# B&R Automation Studio project A2019059_Linka_Power_CP (part 12)

#### Axis_Krokac.st
```iecst
(* TODO: Add your comment here *)
FUNCTION_BLOCK Axis_Krokac

	//***********************************************************Power krokáča*********************************************************************//
	Internal.MC_Power_0.Axis:= AxisName;
	Internal.MC_Power_0.Enable:= CMD.POWER;
	ErrorDetail.Power_Error:= Internal.MC_Power_0.Error;
	ErrorDetail.Power_ErrorID:= Internal.MC_Power_0.ErrorID;
	Internal.MC_Power_0();

	//***********************************************************Zobrazenie stavu krokáča*********************************************************//
	Internal.MC_ReadAxisInfo_0.Axis:= AxisName;
	Internal.MC_ReadAxisInfo_0.Enable:= TRUE;
	STATUS.ReadyToPower_ON := Internal.MC_ReadAxisInfo_0.ReadyForPowerOn;
	STATUS.Communication_READY:= Internal.MC_ReadAxisInfo_0.CommunicationReady;
	STATUS.Power_ON:= Internal.MC_ReadAxisInfo_0.PowerOn;
	STATUS.Homing_OK:= Internal.MC_ReadAxisInfo_0.IsHomed;
	STATUS.EnableSwitch_ACTIVE:= Internal.MC_ReadAxisInfo_0.AdditionalInfo.DigitalInputStatus.DriveEnable;
	STATUS.HomingSwitch_ACTIVE:= Internal.MC_ReadAxisInfo_0.AdditionalInfo.DigitalInputStatus.HomingSwitch;
	STATUS.NegativeLimitSwitch_ACTIVE:=	Internal.MC_ReadAxisInfo_0.AdditionalInfo.DigitalInputStatus.NegativeLimitSwitch;
	STATUS.PositiveLimitSwitch_ACTIVE:=	Internal.MC_ReadAxisInfo_0.AdditionalInfo.DigitalInputStatus.PositiveLimitSwitch;
	Internal.MC_ReadAxisInfo_0();

	//********************************************************Porucha krokáča************************************************************************//
	//Zobrazenie poruchy krokáča//
	Internal.MC_ReadAxisError_0.Axis:= AxisName;
	Internal.MC_ReadAxisError_0.Enable:= CMD.ENABLE;
	STATUS.ERROR_ID:= Internal.MC_ReadAxisError_0.AxisErrorID;
	Internal.MC_ReadAxisError_0();

	Internal.MC_ReadStatus_0.Axis:= AxisName;
	Internal.MC_ReadStatus_0.Enable:= CMD.ENABLE;
	Internal.MC_ReadStatus_0();

	IF Internal.MC_Power_0.Error THEN
		STATUS.ERROR:= TRUE;
	ELSIF Internal.MC_Home_0.Error THEN
		STATUS.ERROR:= TRUE;
	ELSIF Internal.MC_BR_JogLimitPosition_0.Error THEN
		STATUS.ERROR:= TRUE;
	ELSIF Internal.MC_BR_JogVelocity_0.Error THEN
		STATUS.ERROR:= TRUE;
	ELSIF Internal.MC_MoveAbsolute_0.Error THEN
		STATUS.ERROR:= TRUE;
	ELSIF Internal.MC_MoveAdditive_0.Error THEN
		STATUS.ERROR:= TRUE;
	ELSIF Internal.MC_MoveVelocity_0.Error THEN
		STATUS.ERROR:= TRUE;
	ELSIF Internal.MC_Stop_0.Error THEN
		STATUS.ERROR:= TRUE;
	ELSIF Internal.MC_BR_BrakeOperation_0.Error THEN
		STATUS.ERROR:= TRUE;
	ELSIF Internal.MC_BR_InitHome_StpAx_0.Error THEN
		STATUS.ERROR:= TRUE;
	ELSIF STATUS.ERROR_ID <> 0 THEN
		STATUS.ERROR:= TRUE;
	ELSE
		STATUS.ERROR:= FALSE;
	END_IF

	//Reset poruchy krokáča//
	Internal.MC_Reset_0.Axis:= AxisName;
	Internal.MC_Reset_0.Execute:= CMD.ErrorRESET;
	Internal.MC_Reset_0();

	IF CMD.ErrorRESET THEN
		CMD.ENABLE:= FALSE;
	ELSE
		CMD.ENABLE:= TRUE;
	END_IF

	//*********************************************Homing krokáča***************************************************************************//
	//Parametre homingu//
	Internal.MC_BR_InitHome_StpAx_0.Axis:= AxisName;
	Internal.MC_Home_0.Axis:= AxisName;
	IF HomePAR.HomingMode = 0 THEN //Homing na mieste
		Internal.MC_BR_InitHome_StpAx_0.HomingParameters.HomingMode:= mcHOMING_DIRECT;
	ELSIF HomePAR.HomingMode = 1 THEN //Homing na refernčný snímač
		Internal.MC_BR_InitHome_StpAx_0.HomingParameters.HomingMode:= mcHOMING_SWITCH_GATE;
		Internal.MC_BR_InitHome_StpAx_0.HomingParameters.StartDirection:= mcDIR_NEGATIVE;  //Smer hladania refernčného snímača
		Internal.MC_BR_InitHome_StpAx_0.HomingParameters.SwitchEdge:= mcDIR_NEGATIVE; //Typ hrany referenčného snímača
		Internal.MC_BR_InitHome_StpAx_0.HomingParameters.HomingDirection:= mcDIR_POSITIVE; //Smer odchodu z referenčného snímača
	ELSIF HomePAR.HomingMode = 2 THEN //Homing na limitný snímač
		Internal.MC_BR_InitHome_StpAx_0.HomingParameters.HomingMode:= mcHOMING_LIMIT_SWITCH;
		Internal.MC_BR_InitHome_StpAx_0.HomingParameters.SwitchEdge:= mcDIR_NEGATIVE; //Typ hrany referenčného snímača
		Internal.MC_BR_InitHome_StpAx_0.HomingParameters.HomingDirection:= mcDIR_POSITIVE; //Smer odchodu z referenčného snímača
	ELSE
		Internal.MC_BR_InitHome_StpAx_0.HomingParameters.HomingMode:= mcHOMING_DIRECT;
	END_IF
	Internal.MC_BR_InitHome_StpAx_0.HomingParameters.Acceleration:= HomePAR.Acceleration;
	Internal.MC_BR_InitHome_StpAx_0.HomingParameters.HomingVelocity:= HomePAR.HomingVelocity;
	Internal.MC_BR_InitHome_StpAx_0.HomingParameters.Position:= HomePAR.Position;
	Internal.MC_BR_InitHome_StpAx_0.HomingParameters.StartVelocity:= HomePAR.StartVelocity;
	Internal.MC_BR_InitHome_StpAx_0.HomingParameters.ReferencePulse:= mcSWITCH_OFF;
	Internal.MC_BR_InitHome_StpAx_0.HomingParameters.KeepDirection:= mcSWITCH_OFF;
	Internal.MC_Home_0.HomingMode:= mcHOMING_INIT;
	Internal.MC_Home_0.BufferMode:= mcABORTING;
	STATUS.Homing_BUSY:= Internal.MC_Home_0.Busy;
	ErrorDetail.Home_Error:= Internal.MC_Home_0.Error;
	ErrorDetail.Home_ErrorID:= Internal.MC_Home_0.ErrorID;
	Internal.MC_BR_InitHome_StpAx_0();
	Internal.MC_Home_0();

	CASE Internal.Home_STEP OF

		0: //Nulovanie//
			Internal.MC_BR_InitHome_StpAx_0.Execute:= FALSE;
			Internal.MC_Home_0.Execute:= FALSE;
			IF NOT CMD.HOME AND NOT Internal.MC_BR_InitHome_StpAx_0.Error AND NOT Internal.MC_Home_0.Error THEN
				Internal.Home_STEP:= 1;
			END_IF

		1: //Čakanie na spustenie homingu//
			IF CMD.HOME THEN
				Internal.Home_STEP:= 2;
			END_IF

		2: //Načítanie parametrov homingu//
			Internal.MC_BR_InitHome_StpAx_0.Execute:= TRUE;
			IF Internal.MC_BR_InitHome_StpAx_0.Error THEN
				Internal.Home_STEP:= 0;
			ELSIF Internal.MC_BR_InitHome_StpAx_0.Done THEN
				Internal.MC_BR_InitHome_StpAx_0.Execute:= FALSE;
				Internal.Home_STEP:= 3;
			END_IF

		3: //Spustenie homingu
			Internal.MC_Home_0.Execute:= TRUE;
			IF Internal.MC_Home_0.Error THEN
				Internal.Home_STEP:= 0;
			ELSIF Internal.MC_Home_0.Done THEN
				Internal.Home_STEP:= 0;
			ELSIF NOT CMD.HOME THEN
				Internal.Home_STEP:= 0;
			END_IF
	END_CASE

	//*********************************************Jogging krokáča**************************************************************************//

	IF (CMD.JoggVPRED OR CMD.JoggVZAD) AND NOT CMD.JoggLimit_ACTIVE AND CMD.ENABLE THEN
		Internal.MC_BR_JogLimitPosition_0.Enable:= FALSE;
		Internal.MC_BR_JogVelocity_0.Enable:= TRUE;
		STATUS.Jogging_BUSY:= Internal.MC_BR_JogVelocity_0.Jogging;
	ELSIF (CMD.JoggVPRED OR CMD.JoggVZAD) AND CMD.JoggLimit_ACTIVE AND CMD.ENABLE THEN
		Internal.MC_BR_JogVelocity_0.Enable:= FALSE;
		Internal.MC_BR_JogLimitPosition_0.Enable:= TRUE;
		STATUS.Jogging_BUSY:= Internal.MC_BR_JogLimitPosition_0.Jogging;
	ELSE
		Internal.MC_BR_JogVelocity_0.Enable:= FALSE;
		Internal.MC_BR_JogLimitPosition_0.Enable:= FALSE;
	END_IF

	//Normálny jogg//
	Internal.MC_BR_JogVelocity_0.Axis:= AxisName;
	Internal.MC_BR_JogVelocity_0.Acceleration:= PAR.JoggAcceleration;
	Internal.MC_BR_JogVelocity_0.Deceleration:= PAR.JoggDeceleration;
	Internal.MC_BR_JogVelocity_0.Velocity:= PAR.JoggVelocity;
	Internal.MC_BR_JogVelocity_0.Jerk:= 0.0;
	Internal.MC_BR_JogVelocity_0.JogPositive:= CMD.JoggVPRED;
	Internal.MC_BR_JogVelocity_0.JogNegative:= CMD.JoggVZAD;
	ErrorDetail.Jogg_Error:= Internal.MC_BR_JogVelocity_0.Error;
	ErrorDetail.Jogg_ErrorID:= Internal.MC_BR_JogVelocity_0.ErrorID;
	Internal.MC_BR_JogVelocity_0();

	//Limitný jogg//
	Internal.MC_BR_JogLimitPosition_0.Axis:= AxisName;
	IF STATUS.ActualPosition >= PAR.JoggPoziciaLimitVPRED THEN
		Internal.MC_BR_JogLimitPosition_0.LastPosition:= STATUS.ActualPosition;
	ELSE
		Internal.MC_BR_JogLimitPosition_0.LastPosition:= PAR.JoggPoziciaLimitVPRED;
	END_IF
	IF STATUS.ActualPosition <= PAR.JoggPoziciaLimitVZAD THEN
		Internal.MC_BR_JogLimitPosition_0.FirstPosition:= STATUS.ActualPosition;
	ELSE
		Internal.MC_BR_JogLimitPosition_0.FirstPosition:= PAR.JoggPoziciaLimitVZAD;
	END_IF
	Internal.MC_BR_JogLimitPosition_0.Acceleration:= PAR.JoggAcceleration;
	Internal.MC_BR_JogLimitPosition_0.Deceleration:= PAR.JoggDeceleration;
	Internal.MC_BR_JogLimitPosition_0.Jerk:= 0.0;
	Internal.MC_BR_JogLimitPosition_0.JogPositive:= CMD.JoggVPRED;
	Internal.MC_BR_JogLimitPosition_0.JogNegative:= CMD.JoggVZAD;
	Internal.MC_BR_JogLimitPosition_0.Velocity:= PAR.JoggVelocity;
	STATUS.JoggLimit_Dosiahnuty:= Internal.MC_BR_JogLimitPosition_0.LimitReached;
	ErrorDetail.JoggLimit_Error:= Internal.MC_BR_JogLimitPosition_0.Error;
	ErrorDetail.JoggLimit_ErrorID:= Internal.MC_BR_JogLimitPosition_0.ErrorID;
	Internal.MC_BR_JogLimitPosition_0();

	//********************************************Move Absolute***************************************************************************//
	Internal.MC_MoveAbsolute_0.Axis:= AxisName;
	Internal.MC_MoveAbsolute_0.Execute:= CMD.MoveAbsolute;
	Internal.MC_MoveAbsolute_0.Acceleration:= PAR.Acceleration;
	Internal.MC_MoveAbsolute_0.Deceleration:= PAR.Deceleration;
	Internal.MC_MoveAbsolute_0.BufferMode:= mcABORTING;
	IF PAR.MoveDirection = 0 THEN
		Internal.MC_MoveAbsolute_0.Direction:= mcDIR_POSITIVE;
	ELSIF PAR.MoveDirection = 1 THEN
		Internal.MC_MoveAbsolute_0.Direction:= mcDIR_NEGATIVE;
	ELSIF PAR.MoveDirection = 10 THEN
		Internal.MC_MoveAbsolute_0.Direction:= mcDIR_BOTH;
	ELSE
		Internal.MC_MoveAbsolute_0.Direction:= 0;
	END_IF
	Internal.MC_MoveAbsolute_0.Jerk:= 0.0;
	Internal.MC_MoveAbsolute_0.Position:= PAR.Position;
	Internal.MC_MoveAbsolute_0.Velocity:= PAR.Velocity;
	STATUS.MoveAbsolute_BUSY:= Internal.MC_MoveAbsolute_0.Busy;
	STATUS.MoveAbsolute_DONE:= Internal.MC_MoveAbsolute_0.Done;
	ErrorDetail.MoveAbsolute_Error:= Internal.MC_MoveAbsolute_0.Error;
	ErrorDetail.MoveAbsolute_ErrorID:= Internal.MC_MoveAbsolute_0.ErrorID;
	Internal.MC_MoveAbsolute_0();

	//********************************************Move Additive*****************************************************************************//
	Internal.MC_MoveAdditive_0.Axis:= AxisName;
	Internal.MC_MoveAdditive_0.Execute:= CMD.MoveAdditive;
	Internal.MC_MoveAdditive_0.Acceleration:= PAR.Acceleration;
	Internal.MC_MoveAdditive_0.Deceleration:= PAR.Deceleration;
	Internal.MC_MoveAdditive_0.Distance:= PAR.AdditivePosition;
	Internal.MC_MoveAdditive_0.Velocity:= PAR.Velocity;
	Internal.MC_MoveAdditive_0.BufferMode:= mcABORTING;
	Internal.MC_MoveAdditive_0.Jerk:= 0.0;
	STATUS.MoveAdditive_BUSY:= Internal.MC_MoveAdditive_0.Busy;
	STATUS.MoveAdditive_DONE:= Internal.MC_MoveAdditive_0.Done;
	ErrorDetail.MoveAdditive_Error:= Internal.MC_MoveAdditive_0.Error;
	ErrorDetail.MoveAdditive_ErrorID:= Internal.MC_MoveAdditive_0.ErrorID;
	Internal.MC_MoveAdditive_0();

	//*********************************************Move Velocity****************************************************************************//
	Internal.MC_MoveVelocity_0.Axis:= AxisName;
	Internal.MC_MoveVelocity_0.Execute:= CMD.MoveVelocity;
	Internal.MC_MoveVelocity_0.Acceleration:= PAR.Acceleration;
	Internal.MC_MoveVelocity_0.Deceleration:= PAR.Deceleration;
	Internal.MC_MoveVelocity_0.BufferMode:= mcABORTING;
	IF PAR.MoveDirection = 0 THEN
		Internal.MC_MoveVelocity_0.Direction:= mcDIR_POSITIVE;
	ELSIF PAR.MoveDirection = 1 THEN
		Internal.MC_MoveVelocity_0.Direction:= mcDIR_NEGATIVE;
	ELSIF PAR.MoveDirection = 10 THEN
		Internal.MC_MoveVelocity_0.Direction:= mcDIR_BOTH;
	ELSE
		Internal.MC_MoveVelocity_0.Direction:= 0;
	END_IF
	Internal.MC_MoveVelocity_0.Velocity:= PAR.Velocity;
	Internal.MC_MoveVelocity_0.Jerk:= 0.0;
	STATUS.MoveVelocity_BUSY:= Internal.MC_MoveVelocity_0.Busy;
	STATUS.Rychlost_Dosiahnuta:= Internal.MC_MoveVelocity_0.InVelocity;
	ErrorDetail.MoveVelocity_Error:= Internal.MC_MoveVelocity_0.Error;
	ErrorDetail.MoveVelocity_ErrorID:= Internal.MC_MoveVelocity_0.ErrorID;
	Internal.MC_MoveVelocity_0();

	//********************************************Stop krokáča******************************************************************************//
	Internal.MC_Stop_0.Axis:= AxisName;
	Internal.MC_Stop_0.Execute:= CMD.STOP;
	Internal.MC_Stop_0.Deceleration:= PAR.StopDeceleration;
	Internal.MC_Stop_0.Jerk:= 0.0;
	STATUS.STOP_ACTIVE:= Internal.MC_Stop_0.Done;
	ErrorDetail.Stop_Error:= Internal.MC_Stop_0.Error;
	ErrorDetail.Stop_ErrorID:= Internal.MC_Stop_0.ErrorID;
	Internal.MC_Stop_0();

	//**********************************************Ovládanie brzdy************************************************************************//
	Internal.MC_BR_BrakeOperation_0.Axis:= AxisName;
	IF CMD.UvolniBRZDU THEN
		Internal.MC_BR_BrakeOperation_0.Command:= mcBRAKE_OPEN;
		Internal.MC_BR_BrakeOperation_0.Execute:= TRUE;
		STATUS.UvolnenieBrzdy_DONE:= Internal.MC_BR_BrakeOperation_0.Done;
	ELSIF CMD.ZabrzdiBRZDU THEN
		Internal.MC_BR_BrakeOperation_0.Command:= mcBRAKE_CLOSE;
		Internal.MC_BR_BrakeOperation_0.Execute:= TRUE;
		STATUS.ZabrzdenieBrzdy_DONE:= Internal.MC_BR_BrakeOperation_0.Done;
	ELSE
		Internal.MC_BR_BrakeOperation_0.Execute:= FALSE;
		STATUS.UvolnenieBrzdy_DONE:= FALSE;
		STATUS.ZabrzdenieBrzdy_DONE:= FALSE;
	END_IF
	ErrorDetail.BreakOperation_Error:= Internal.MC_BR_BrakeOperation_0.Error;
	ErrorDetail.BreakOperation_ErrorID:= Internal.MC_BR_BrakeOperation_0.ErrorID;
	Internal.MC_BR_BrakeOperation_0();

	//**********************************************Aktuálna pozícia*************************************************************************//
	Internal.MC_ReadActualPosition_0.Axis:= AxisName;
	Internal.MC_ReadActualPosition_0.Enable:= CMD.ENABLE;
	STATUS.ActualPosition:=	Internal.MC_ReadActualPosition_0.Position;
	Internal.MC_ReadActualPosition_0();

	//**********************************************Aktuálna rýchlosť*************************************************************************//
	Internal.MC_ReadActualVelocity_0.Axis:= AxisName;
	Internal.MC_ReadActualVelocity_0.Enable:= CMD.ENABLE;
	STATUS.ActualVelocity:= Internal.MC_ReadActualVelocity_0.Velocity;
	Internal.MC_ReadActualVelocity_0();

	//*********************************************Zmena rýchlosti a rampy********************************************************************//
	Internal.MC_SetOverride_0.Axis:= AxisName;
	Internal.MC_SetOverride_0.Enable:= CMD.UpdatePAR;
	IF PAR.ZmenaRampy < 0.1 THEN
		Internal.MC_SetOverride_0.AccFactor:= 0.1;
	ELSIF PAR.ZmenaRampy > 2.0 THEN
		Internal.MC_SetOverride_0.AccFactor:= 2.0;
	ELSE
		Internal.MC_SetOverride_0.AccFactor:= PAR.ZmenaRampy;
	END_IF
	IF PAR.ZmenaRychlosti < 0.1 THEN
		Internal.MC_SetOverride_0.VelFactor:= 0.1;
	ELSIF PAR.ZmenaRychlosti > 2.0 THEN
		Internal.MC_SetOverride_0.VelFactor:= 2.0;
	ELSE
		Internal.MC_SetOverride_0.VelFactor:= PAR.ZmenaRychlosti;
	END_IF
	STATUS.UpdatePAR_DONE:= Internal.MC_SetOverride_0.Enabled;
	Internal.MC_SetOverride_0();

END_FUNCTION_BLOCK
```

#### ServoLim.st
```iecst
(* TODO: Add your comment here *)
FUNCTION_BLOCK ServoLim

	//*******************************Aktivácia limitných snímačov*****************************************//
	//Reset poruchy//
	IF NOT ENABLE THEN
		Internal.STEP:= 0;
		Error:= FALSE;
	END_IF

	//Zápis do parametrov//

	CASE Internal.STEP OF

		0: //Čakanie na spustenie sekvencie//
			Internal.MC_BR_ProcessParID_AcpAx_0.Execute:= FALSE;
			Internal.MC_BR_CyclicProcessParID_AcpAx_0.Enable:= FALSE;
			BUSY:= FALSE;
			IF ENABLE AND NOT Error THEN
				Internal.STEP:= 1;
			END_IF

		1://Zápis parametru - povolenie limitných snímačov//
			Internal.MC_BR_ProcessParID_AcpAx_0.Axis:= AxisName;
			Internal.MC_BR_ProcessParID_AcpAx_0.DataAddress:= ADR(Internal.McAcpAxProcessParIDType_0);
			Internal.MC_BR_ProcessParID_AcpAx_0.NumberOfParIDs:= 0;
			Internal.MC_BR_ProcessParID_AcpAx_0.Mode:= mcACPAX_PARID_SET;
			Internal.McAcpAxProcessParIDType_0.DataType:= mcACPAX_PARTYPE_USINT;
			Internal.McAcpAxProcessParIDType_0.ParID:= 184;
			Internal.McAcpAxProcessParIDType_0.VariableAddress:= ADR(Internal.AktivaciaLimSnimacov_Data);
			Internal.AktivaciaLimSnimacov_Data:= 7;
			Internal.MC_BR_ProcessParID_AcpAx_0.Execute:= TRUE;

			IF Internal.MC_BR_ProcessParID_AcpAx_0.Done THEN
				Internal.MC_BR_ProcessParID_AcpAx_0.Execute:= FALSE;
				Internal.AktivaciaLimSnimacov_Data:= 0;
				Internal.STEP:= 3;
			ELSIF Internal.MC_BR_ProcessParID_AcpAx_0.Error THEN
				Error:= TRUE;
				Internal.STEP:= 0;
			END_IF

		3://Korekčný čas//
			IF NOT Internal.MC_BR_ProcessParID_AcpAx_0.Done THEN
				Internal.KorekcnyCas.IN:= TRUE;
			END_IF

			IF Internal.KorekcnyCas.Q THEN
				Internal.KorekcnyCas.IN:= FALSE;
				Internal.STEP:= 5;
			END_IF

		5://Čítanie parametru - overenie povolenia limitných snímačov//
			Internal.MC_BR_ProcessParID_AcpAx_0.Axis:= AxisName;
			Internal.MC_BR_ProcessParID_AcpAx_0.DataAddress:= ADR(Internal.McAcpAxProcessParIDType_0);
			Internal.MC_BR_ProcessParID_AcpAx_0.NumberOfParIDs:= 0;
			Internal.MC_BR_ProcessParID_AcpAx_0.Mode:= mcACPAX_PARID_GET;
			Internal.McAcpAxProcessParIDType_0.DataType:= mcACPAX_PARTYPE_USINT;
			Internal.McAcpAxProcessParIDType_0.ParID:= 184;
			Internal.McAcpAxProcessParIDType_0.VariableAddress:= ADR(Internal.AktivaciaLimSnimacov_Data);
			Internal.MC_BR_ProcessParID_AcpAx_0.Execute:= TRUE;

			IF Internal.MC_BR_ProcessParID_AcpAx_0.Done THEN
				IF Internal.AktivaciaLimSnimacov_Data = 7 THEN
					Internal.MC_BR_ProcessParID_AcpAx_0.Execute:= FALSE;
					Internal.STEP:= 10;
				ELSE
					Error:= TRUE;
					Internal.STEP:= 0;
				END_IF
			ELSIF Internal.MC_BR_ProcessParID_AcpAx_0.Error THEN
				Error:= TRUE;
				Internal.STEP:= 0;
			END_IF

		8://Korekčný čas//
			IF NOT Internal.MC_BR_ProcessParID_AcpAx_0.Done THEN
				Internal.KorekcnyCas.IN:= TRUE;
			END_IF

			IF Internal.KorekcnyCas.Q THEN
				Internal.KorekcnyCas.IN:= FALSE;
				Internal.STEP:= 10;
			END_IF

		10://
			Internal.MC_BR_CyclicProcessParID_AcpAx_0.Axis:= AxisName;
			Internal.MC_BR_CyclicProcessParID_AcpAx_0.DataAddress:= ADR(Internal.McAcpAxCycParIDType_0);
			Internal.MC_BR_CyclicProcessParID_AcpAx_0.NumberOfParIDs:= 0;
			Internal.MC_BR_CyclicProcessParID_AcpAx_0.Mode:= mcACPAX_CYCLIC_PARID_WRITE;
			Internal.McAcpAxCycParIDType_0.DataType:= mcACPAX_PARTYPE_USINT;
			Internal.McAcpAxCycParIDType_0.ParID:= 185;
			Internal.McAcpAxCycParIDType_0.VariableAddress:= ADR(Internal.LimSnimace_Data);
			Internal.McAcpAxCycParIDType_0.RefreshMode:= mcACPAX_CYCLIC_EVERY_RECORD;
			Internal.MC_BR_CyclicProcessParID_AcpAx_0.Enable:= TRUE;
			Internal.LimSnimace_Data.0:= HomingSwitch;
			Internal.LimSnimace_Data.1:= PositiveLimitSwitch;
			Internal.LimSnimace_Data.2:= NegativeLimitSwitch;

			BUSY:= Internal.MC_BR_CyclicProcessParID_AcpAx_0.Busy;

			IF Internal.MC_BR_CyclicProcessParID_AcpAx_0.Error THEN
				Error:= TRUE;
				Internal.STEP:= 0;
			END_IF

	END_CASE

	Internal.MC_BR_ProcessParID_AcpAx_0();
	Internal.MC_BR_CyclicProcessParID_AcpAx_0();

	Internal.KorekcnyCas.PT:= T#200ms;
	Internal.KorekcnyCas();

END_FUNCTION_BLOCK
```

### Library Logical/Libraries/IecCheck (IEC)
Depends on: sys_lib, AsBrStr

#### IecCheck.fun - Exported functions and function blocks
```iecst
FUNCTION CheckDivSint : SINT (* Check divisor for SINT division *)
	VAR_INPUT
		divisor : SINT;
	END_VAR
END_FUNCTION

FUNCTION CheckDivUsint : USINT (* Check divisor for USINT division *)
	VAR_INPUT
		divisor : USINT;
	END_VAR
END_FUNCTION

FUNCTION CheckDivInt : INT (* Check divisor for INT division *)
	VAR_INPUT
		divisor : INT;
	END_VAR
END_FUNCTION

FUNCTION CheckDivUint : UINT (* Check divisor for UINT division *)
	VAR_INPUT
		divisor : UINT;
	END_VAR
END_FUNCTION

FUNCTION CheckDivDint : DINT (* Check divisor for DINT division *)
	VAR_INPUT
		divisor : DINT;
	END_VAR
END_FUNCTION

FUNCTION CheckDivUdint : UDINT (* Check divisor for UDINT division *)
	VAR_INPUT
		divisor : UDINT;
	END_VAR
END_FUNCTION

FUNCTION CheckDivReal : REAL (* Check divisor for REAL division *)
	VAR_INPUT
		divisor : REAL;
	END_VAR
END_FUNCTION

FUNCTION CheckDivLReal : LREAL (* Check divisor for LREAL division, not available for SG3 and SGC *)
	VAR_INPUT
		divisor : LREAL;
	END_VAR
END_FUNCTION

FUNCTION CheckBounds : DINT (* Check range for array access *)
	VAR_INPUT
		index : DINT;
		lower : DINT;
		upper : DINT;
	END_VAR
END_FUNCTION

FUNCTION CheckRange : DINT (* Check range for enumeration *)
	VAR_INPUT
		value : DINT;
		lower : DINT;
		upper : DINT;
	END_VAR
END_FUNCTION

FUNCTION CheckSignedSubrange : DINT (* Check range for subrange of signed data types *)
	VAR_INPUT
		value : DINT;
		lower : DINT;
		upper : DINT;
	END_VAR
END_FUNCTION

FUNCTION CheckUnsignedSubrange : UDINT (* Check range for subrange of unsigned data types *)
	VAR_INPUT
		value : UDINT;
		lower : UDINT;
		upper : UDINT;
	END_VAR
END_FUNCTION

FUNCTION CheckReadAccess : UDINT (* Check address when reading dynamic variables *)
	VAR_INPUT
		address : UDINT;
	END_VAR
END_FUNCTION

FUNCTION CheckWriteAccess : UDINT (* Check address when writing dynamic variables *)
	VAR_INPUT
		address : UDINT;
	END_VAR
END_FUNCTION

FUNCTION MakeEntry : UDINT (* Makes an entry (log book entry) in the error log book *)
	VAR
		taskname : STRING[30];
		group : USINT;
		status_name : UINT;
		out_text : STRING[80];
	END_VAR
	VAR_INPUT
		number : UINT;
		index : DINT;
		text : STRING[50];
	END_VAR
END_FUNCTION
```

#### IecCheck.st - Implementation file
```iecst
(* Check divisor for SINT division *)
FUNCTION CheckDivSint
	IF divisor=0 THEN
		CheckDivSint:=1;
		MakeEntry(55555,divisor,'CheckDivSint');
	ELSE
		CheckDivSint:=divisor;
	END_IF
END_FUNCTION

(* Check divisor for USINT division *)
FUNCTION CheckDivUsint
	IF divisor=0 THEN
		CheckDivUsint:=1;
		MakeEntry(55555,divisor,'CheckDivUsint');
	ELSE
		CheckDivUsint:=divisor;
	END_IF
END_FUNCTION

(* Check divisor for INT division *)
FUNCTION CheckDivInt
	IF divisor=0 THEN
		CheckDivInt:=1;
		MakeEntry(55555,divisor,'CheckDivInt');
	ELSE
		CheckDivInt:=divisor;
	END_IF
END_FUNCTION

(* Check divisor for UINT division *)
FUNCTION CheckDivUint
	IF divisor=0 THEN
		CheckDivUint:=1;
		MakeEntry(55555,divisor,'CheckDivUint');
	ELSE
		CheckDivUint:=divisor;
	END_IF
END_FUNCTION

(* Check divisor for DINT division *)
FUNCTION CheckDivDint
	IF divisor=0 THEN
		CheckDivDint:=1;
		MakeEntry(55555,divisor,'CheckDivDint');
	ELSE
		CheckDivDint:=divisor;
	END_IF
END_FUNCTION

(* Check divisor for UDINT division *)
FUNCTION CheckDivUdint
	IF divisor=0 THEN
		CheckDivUdint:=1;
		MakeEntry(55555,divisor,'CheckDivUdint');
	ELSE
		CheckDivUdint:=divisor;
	END_IF
END_FUNCTION

(* Check divisor for REAL division *)
FUNCTION CheckDivReal
	IF divisor=0 THEN
		CheckDivReal:=1;
		MakeEntry(55555,0,'CheckDivReal');
	ELSE
		CheckDivReal:=divisor;
	END_IF
END_FUNCTION

(* Check divisor for LREAL division *)
FUNCTION CheckDivLReal
	IF divisor=0 THEN
		CheckDivLReal:=1;
		MakeEntry(55555,0,'CheckDivLReal');
	ELSE
		CheckDivLReal:=divisor;
	END_IF
END_FUNCTION

(* Check range for array access *)
FUNCTION CheckBounds
	IF index < lower THEN
		CheckBounds := lower;
		MakeEntry(55555,index,'CheckBounds');
	ELSIF index > upper THEN
		CheckBounds := upper;
		MakeEntry(55555,index,'CheckBounds');
	ELSE
		CheckBounds := index;
	END_IF
END_FUNCTION

(* Check range for enumeration *)
FUNCTION CheckRange
	IF value < lower THEN
		CheckRange := lower;
		MakeEntry(55555,value,'CheckRange');
	ELSIF value > upper THEN
		CheckRange := upper;
		MakeEntry(55555,value,'CheckRange');
	ELSE
		CheckRange := value;
	END_IF
END_FUNCTION

(* Check range for subrange of signed data types *)
FUNCTION CheckSignedSubrange
	IF value < lower THEN
		CheckSignedSubrange := lower;
		MakeEntry(55555,value,'CheckSignedSubrange');
	ELSIF value > upper THEN
		CheckSignedSubrange := upper;
		MakeEntry(55555,value,'CheckSignedSubrange');
	ELSE
		CheckSignedSubrange := value;
	END_IF
END_FUNCTION

(* Check range for subrange of unsigned data types *)
FUNCTION CheckUnsignedSubrange
	IF value < lower THEN
		CheckUnsignedSubrange := lower;
		MakeEntry(55555,value,'CheckUnsignedSubrange');
	ELSIF value > upper THEN
		CheckUnsignedSubrange := upper;
		MakeEntry(55555,value,'CheckUnsignedSubrange');
	ELSE
		CheckUnsignedSubrange := value;
	END_IF
END_FUNCTION

(* Check address when reading dynamic variables *)
FUNCTION CheckReadAccess
	IF address=0 THEN
		(* TODO: Insert an appropriate code, see AutomationStudio help for further information *)
		MakeEntry(55555,address,'Read from NULL');
	END_IF

	CheckReadAccess:=0;
END_FUNCTION

(* Check address when writing dynamic variables *)
FUNCTION CheckWriteAccess
	IF address=0 THEN
		(* TODO: Insert an appropriate code, see AutomationStudio help for further information *)
		MakeEntry(55555,address,'Write to NULL');
	END_IF

	CheckWriteAccess:=0;
END_FUNCTION

(* Makes an entry (log book entry) in the error log book *)
FUNCTION MakeEntry
		status_name := ST_name(0,ADR(taskname),ADR(group));

		brsstrcpy(ADR(out_text),ADR(text));
		brsstrcat(ADR(out_text),ADR(' > in task > '));
  		brsstrcat(ADR(out_text),ADR(taskname));
		MakeEntry := ADR(out_text);
		ERRxwarning(number,index,ADR(out_text));
END_FUNCTION
```

### Library Logical/Libraries/AtlasCopco (IEC)

#### AtlasCopco.fun - Exported functions and function blocks
```iecst
{REDUND_ERROR} FUNCTION_BLOCK PrevodMomentu (*TODO: Prevod momentu s menicov atlas copco*) (*$GROUP=User,$CAT=User,$GROUPICON=User.png,$CATICON=User.png*)
	VAR_INPUT
		AtlasMaximalnaTolerancia : UDINT;
		AtlasMinimalnaTolerancia : UDINT;
		AtlasAktualnyMoment : UDINT;
	END_VAR
	VAR_OUTPUT
		ToleranciaMAX : REAL;
		ToleranciaMIN : REAL;
		AktualnyMoment : REAL;
	END_VAR
	VAR
		ByteArray2 : ARRAY[0..3] OF USINT;
		ByteArray3 : ARRAY[0..3] OF USINT;
		ByteArray1 : ARRAY[0..3] OF USINT;
		InputShifted2 : UDINT;
		InputShifted3 : UDINT;
		InputShifted1 : UDINT;
		Index2 : USINT;
		Index3 : USINT;
		Index1 : USINT;
	END_VAR
END_FUNCTION_BLOCK

{REDUND_ERROR} {REDUND_UNREPLICABLE} FUNCTION_BLOCK Round (*Zaokrúhlenie na jedno desatinné miesto*) (*$GROUP=User,$CAT=User,$GROUPICON=User.png,$CATICON=User.png*)
	VAR_INPUT
		VstupnaHodnota : {REDUND_UNREPLICABLE} UINT;
	END_VAR
	VAR_OUTPUT
		VystupnaHodnota : {REDUND_UNREPLICABLE} REAL;
	END_VAR
	VAR
		VstupnaHodnotaREAL : {REDUND_UNREPLICABLE} REAL;
		VysledokDeleniaUINT : {REDUND_UNREPLICABLE} UINT;
		VysledokDeleniaREAL : {REDUND_UNREPLICABLE} REAL;
	END_VAR
END_FUNCTION_BLOCK
```

#### PrevodMomentu.st
```iecst
(* TODO: Prevod momentu z menicov atlas copco *)
FUNCTION_BLOCK PrevodMomentu

//aktualny moment
		//rozbitie UDINT na pole USINTov
    InputShifted1:=AtlasAktualnyMoment;

    FOR Index1:=0 TO 3 DO
        ByteArray1[Index1]:=UDINT_TO_USINT(InputShifted1);
        InputShifted1:=ROR(InputShifted1,8);
    END_FOR

    //spojenie USINT do REAL vo vhodnej forme ;-)
    AktualnyMoment:=ByteArray1[3]*0.01+ByteArray1[1];

    //tolerancia MIN
    //rozbitie UDINT na pole USINTov
    InputShifted2:=AtlasMinimalnaTolerancia;

    FOR Index2:=0 TO 3 DO
        ByteArray2[Index2]:=UDINT_TO_USINT(InputShifted2);
        InputShifted2:=ROR(InputShifted2,8);
    END_FOR

    //spojenie USINT do REAL vo vhodnej forme ;-)
    ToleranciaMIN:=ByteArray2[3]*0.01+ByteArray2[1];

    //tolerancia MAX
    //rozbitie UDINT na pole USINTov
    InputShifted3:=AtlasMaximalnaTolerancia;

    FOR Index3:=0 TO 3 DO
        ByteArray3[Index3]:=UDINT_TO_USINT(InputShifted3);
        InputShifted3:=ROR(InputShifted3,8);
    END_FOR

    //spojenie USINT do REAL vo vhodnej forme ;-)
    ToleranciaMAX:=ByteArray3[3]*0.01+ByteArray3[1];
END_FUNCTION_BLOCK
```

#### Round.st - Zaokruhlenie hodnoty vysunutia srobovacky
```iecst
(* Zaokrúhlenie na jedno desatinné miesto *)
FUNCTION_BLOCK Round

    VstupnaHodnotaREAL:= UINT_TO_REAL(VstupnaHodnota);
    IF VstupnaHodnotaREAL >= 128 THEN
        VysledokDeleniaUINT:= TRUNC((VstupnaHodnotaREAL /128)*10);
        VysledokDeleniaREAL:= UINT_TO_REAL(VysledokDeleniaUINT);
        VystupnaHodnota:= VysledokDeleniaREAL /10;
    ELSE
        VystupnaHodnota:= 0;
    END_IF

END_FUNCTION_BLOCK
```

### Library Logical/Libraries/SKTcp (ANSIC, version 1.00.8) - Panasonic TCP Client Traceabilita
Depends on: AsBrStr, AsTCP, sys_lib, standard, IecCheck, FileIO

#### Types.typ - Exported data types
```iecst
(*

         projekt: SKTcp - Panasonic

         autor: Ing. Milan Jun
         company: B+R Automatizace spol. s r.o.
         date: 10.09.2020

*)

TYPE
	SKTcpClientSC_Type : 	STRUCT
		StepName : STRING[255];
		bNext : BOOL;
		bJump : BOOL;
		bLast : BOOL;
		bRepeat : BOOL;
		edge : BOOL;
		step : UINT;
		idle_time : TON;
		alarm_time : TON;
	END_STRUCT;
END_TYPE

(**)

TYPE
	SKTcpClientTraceStatus_Type : 	STRUCT
		RecvSize : UDINT;
		DataRecv : ARRAY[0..4999]OF USINT;
		RecvCounter : UDINT;
		enaSend : BOOL;
		staReceived : BOOL;
		staSent : BOOL;
		staError : BOOL;
		staErrorSent : BOOL;
		staErrorOpen : BOOL;
		staErrorRecv : BOOL;
		staErrorIoctl : BOOL;
		staErrorClose : BOOL;
		staErrorClient : BOOL;
		staErrorRecvTout : BOOL;
		staErrorConn : BOOL;
		staErrorConnTout : BOOL;
		staSending : BOOL;
		staReceiving : BOOL;
		staReadyToClose : BOOL;
		staReadyToSend : BOOL;
	END_STRUCT;
	SKTcpClientTraceParPackInter_Typ : 	STRUCT
		start : USINT;
		length_int : UINT;
		length_str : STRING[5];
		xor : BYTE;
		xor_str : USINT;
		stop : USINT;
		ti : USINT;
		length : UINT;
		ret_len : UINT;
	END_STRUCT;
	SKTcpClientTraceParams_Type : 	STRUCT
		IPaddrServ : ARRAY[0..39]OF USINT;
		IPportClient : UINT;
		IPportServ : UINT;
		disRecv : BOOL;
		enaClose : BOOL; (*Zatvorenie portu po prijati odpovede od servera*)
		RecvTimeout : UDINT := 3000;
		ConnTimeout : UDINT := 3000;
		Packet : SKTcpClientTraceParamsPack_Typ;
	END_STRUCT;
	SKTcpClientTraceParamsPack_Typ : 	STRUCT
		internal : SKTcpClientTraceParPackInter_Typ;
		type : STRING[1];
		workplace : STRING[5];
		rfid : STRING[10];
		master : STRING[30];
		dps1 : STRING[30];
		dps2 : STRING[30];
		dps3 : STRING[30];
		dps4 : STRING[30];
		dps5 : STRING[30];
		operator_id : STRING[8];
		data_report : STRING[4000];
		result : STRING[4];
	END_STRUCT;
	SKTcpClientTraceLogger_Typ : 	STRUCT
		LastDataRecv : STRING[5000];
		LastDataSend : STRING[5000];
		SLOGGER : ARRAY[0..99]OF STRING[5000];
		RLOGGER : ARRAY[0..99]OF STRING[5000];
	END_STRUCT;
	SKTcpClientTraceIntern_Type : 	STRUCT
		Step : UINT;
		Ident : UDINT;
		TCP_Open : TcpOpen;
		TCP_Close : TcpClose;
		TCP_Client : TcpClient;
		TCP_Recv : TcpRecv;
		TCP_Send : TcpSend;
		TCP_Ioctl : TcpIoctl;
		linger_opt : tcpLINGER_typ;
		TimerRecv : TON;
		TimerConn : TON;
		cmdClose : BOOL;
		cmdSend : BOOL;
		CloseOld : BOOL;
		SendOld : BOOL;
		EnableOld : BOOL;
		Splitter : SKTcpClientSplitter;
		oneskorenie : TON;
	END_STRUCT;
	SKTcpClientTraceDataSend_Type : 	STRUCT
		send_data_a : ARRAY[0..4999]OF USINT;
		send_data_b : ARRAY[0..4999]OF USINT;
		DataSend : ARRAY[0..4999]OF USINT;
	END_STRUCT;
	SKTcpClientTraceCmd_Type : 	STRUCT
		Send : BOOL;
		Close : BOOL;
	END_STRUCT;
	SKTcpClientTestParPackInter_Type : 	STRUCT
		start : USINT;
		data_length : UINT;
		length : USINT;
		xor : USINT;
		stop : USINT;
		ti : USINT;
	END_STRUCT;
END_TYPE

(**)

TYPE
	SKTcpClientTesterStatus_Type : 	STRUCT
		RecvSize : UDINT;
		DataRecv : ARRAY[0..199]OF USINT;
		RecvCounter : UDINT;
		enaSend : BOOL;
		staReceived : BOOL;
		staSent : BOOL;
		staError : BOOL;
		staErrorSent : BOOL;
		staErrorOpen : BOOL;
		staErrorRecv : BOOL;
		staErrorIoctl : BOOL;
		staErrorClose : BOOL;
		staErrorClient : BOOL;
		staErrorRecvTout : BOOL;
		staErrorConn : BOOL;
		staErrorConnTout : BOOL;
		staSending : BOOL;
		staReceiving : BOOL;
		staReadyToClose : BOOL;
		staReadyToSend : BOOL;
	END_STRUCT;
	SKTcpClientTesterParams_Type : 	STRUCT
		IPaddrServ : ARRAY[0..39]OF USINT;
		IPportClient : UINT;
		IPportServ : UINT;
		disRecv : BOOL;
		enaClose : BOOL; (*Zatvorenie portu po prijati odpovede od servera*)
		RecvTimeout : UDINT := 3000;
		ConnTimeout : UDINT := 3000;
		Packet : SKTcpClientTesterParamsPack_Type;
	END_STRUCT;
	SKTcpClientTesterParamsPack_Type : 	STRUCT
		type : USINT;
		workplace : USINT;
		id : USINT;
		data : ARRAY[0..31]OF USINT;
		internal : SKTcpClientTestParPackInter_Type;
	END_STRUCT;
	SKTcpClientTesterLogger_Typ : 	STRUCT
		LastDataRecv : STRING[2000];
		LastDataSend : STRING[2000];
		SLOGGER : ARRAY[0..99]OF STRING[2000];
		RLOGGER : ARRAY[0..99]OF STRING[2000];
	END_STRUCT;
	SKTcpClientTesterIntern_Type : 	STRUCT
		Step : UINT;
		Ident : UDINT;
		TCP_Open : TcpOpen;
		TCP_Close : TcpClose;
		TCP_Client : TcpClient;
		TCP_Recv : TcpRecv;
		TCP_Send : TcpSend;
		TCP_Ioctl : TcpIoctl;
		linger_opt : tcpLINGER_typ;
		TimerRecv : TON;
		TimerConn : TON;
		cmdClose : BOOL;
		cmdSend : BOOL;
		CloseOld : BOOL;
		SendOld : BOOL;
		EnableOld : BOOL;
	END_STRUCT;
	SKTcpClientTesterDataSend_Type : 	STRUCT
		SendLength : UDINT;
		send_data_a : ARRAY[0..199]OF USINT;
		DataSend : ARRAY[0..199]OF USINT;
	END_STRUCT;
	SKTcpClientTesterCmd_Type : 	STRUCT
		Send : BOOL;
		Close : BOOL;
	END_STRUCT;
END_TYPE

(**)

TYPE
	SKTcpClientFtpParamSrc_Typ : 	STRUCT
		pDevice : UDINT;
		pParam : UDINT;
		pPath : UDINT;
	END_STRUCT;
	SKTcpClientFtpParamDest_Typ : 	STRUCT
		pDevice : UDINT;
		pParam : UDINT;
		pPath : UDINT;
		pNewName : UDINT;
	END_STRUCT;
	SKTcpClientFtpParam_Typ : 	STRUCT
		src : SKTcpClientFtpParamSrc_Typ;
		dest : SKTcpClientFtpParamDest_Typ;
	END_STRUCT;
	SKTcpClientFtpInternal_Typ : 	STRUCT
		fb : SKTcpClientFtpInternalFb_Typ;
		sc : SKTcpClientSC_Type;
		src_handle : UDINT;
		dest_handle : UDINT;
	END_STRUCT;
	SKTcpClientFtpInternalFb_Typ : 	STRUCT
		Devlink_0 : DevLink;
		DevUnlink_0 : DevUnlink;
		FileInfo_0 : FileInfo;
		DirInfo_0 : DirInfo;
		FileRename_0 : FileRename;
		DirRead_0 : DirRead;
		FileCopy_0 : FileCopy;
		FileDelete_0 : FileDelete;
	END_STRUCT;
	SKTcpClientFtpStatusSrc_Typ : 	STRUCT
		pData : fiDIR_READ_DATA;
	END_STRUCT;
	SKTcpClientFtpStatusDest_Typ : 	STRUCT
		empty : USINT;
	END_STRUCT;
	SKTcpClientFtpStatus_Typ : 	STRUCT
		src : SKTcpClientFtpStatusSrc_Typ;
		dest : SKTcpClientFtpStatusDest_Typ;
	END_STRUCT;
END_TYPE
```

#### Constants.var - Exported constants
```iecst
(*

         projekt: SKTcp - Panasonic

         autor: Ing. Milan Jun
         company: B+R Automatizace spol. s r.o.
         date: 10.09.2020

*)
VAR CONSTANT
	MAX_CHARACTER : UINT := 1;
	MAX_STRING : UINT := 5000;
	MAX_STRING_MINUS_ONE : UINT := 4999;
END_VAR
(**)
VAR CONSTANT
	MAX_TRACE_LOGGER_ENTIRES : USINT := 90;
END_VAR
```

#### SKTcp.fun - Exported functions and function blocks
```iecst
(**************************************************************

         projekt: SKTcp - Panasonic

         autor: Ing. Milan Jun
         company: B+R Automatizace spol. s r.o.
         date: 10.09.2020

*)

{REDUND_ERROR} FUNCTION_BLOCK SKTcpClientSplitter (*SKTcpClient - Splitter*) (*$GROUP=User,$CAT=User,$GROUPICON=User.png,$CATICON=User.png*)
	VAR_INPUT
		enable : BOOL;
		iSelector : USINT;
		iInputString : STRING[MAX_STRING];
	END_VAR
	VAR_OUTPUT
		out : ARRAY[0..14] OF STRING[MAX_STRING];
		done : BOOL;
		OUT_Master : STRING[30];
		OUT_Typ : STRING[1];
		OUT_Result : STRING[2];
	END_VAR
	VAR
		enableOld : BOOL;
		tmpInputString : ARRAY[0..MAX_STRING_MINUS_ONE] OF USINT;
		tmpString : STRING[MAX_CHARACTER];
		idx : ARRAY[0..1] OF UDINT;
	END_VAR
END_FUNCTION_BLOCK

{REDUND_ERROR} FUNCTION_BLOCK SKTcpClientTester (*SKTcpClient - Tester*) (*$GROUP=User,$CAT=User,$GROUPICON=User.png,$CATICON=User.png*)
	VAR_INPUT
		Enable : BOOL;
		Cmd : SKTcpClientTesterCmd_Type;
		Params : SKTcpClientTesterParams_Type;
		DataSend : SKTcpClientTesterDataSend_Type;
	END_VAR
	VAR_OUTPUT
		Status : SKTcpClientTesterStatus_Type;
		FBStatus : {REDUND_UNREPLICABLE} UINT;
		logger : SKTcpClientTesterLogger_Typ;
	END_VAR
	VAR
		Internal : SKTcpClientTesterIntern_Type;
	END_VAR
END_FUNCTION_BLOCK

{REDUND_ERROR} FUNCTION_BLOCK SKTcpClientTrace (*SKTcpClient - ZberDat verzia 2*) (*$GROUP=User,$CAT=User,$GROUPICON=User.png,$CATICON=User.png*)
	VAR_INPUT
		Enable : BOOL;
		Cmd : SKTcpClientTraceCmd_Type;
		Params : SKTcpClientTraceParams_Type;
		DataSend : SKTcpClientTraceDataSend_Type;
	END_VAR
	VAR_OUTPUT
		Status : SKTcpClientTraceStatus_Type;
		FBStatus : {REDUND_UNREPLICABLE} UINT;
		logger : SKTcpClientTraceLogger_Typ;
	END_VAR
	VAR
		Internal : SKTcpClientTraceIntern_Type;
	END_VAR
END_FUNCTION_BLOCK

{REDUND_ERROR} FUNCTION_BLOCK SKTcpClientEdge (*SKTcpClient - Edge*) (*$GROUP=User,$CAT=User,$GROUPICON=User.png,$CATICON=User.png*)
	VAR_INPUT
		CLK : BOOL;
	END_VAR
	VAR_OUTPUT
		Q : {REDUND_UNREPLICABLE} BOOL;
	END_VAR
	VAR
		Last_State : BOOL;
	END_VAR
END_FUNCTION_BLOCK

{REDUND_ERROR} FUNCTION_BLOCK SKTcpClientFTP (*SKTcpClient - FTP*) (*$GROUP=User,$CAT=User,$GROUPICON=User.png,$CATICON=User.png*)
	VAR_INPUT
		enable : BOOL;
		send : BOOL;
		param : SKTcpClientFtpParam_Typ;
	END_VAR
	VAR_OUTPUT
		active : BOOL;
		status : SKTcpClientFtpStatus_Typ;
		Errorcode : UINT;
	END_VAR
	VAR
		internal : SKTcpClientFtpInternal_Typ;
	END_VAR
END_FUNCTION_BLOCK

{REDUND_ERROR} FUNCTION SKTcpClientNod : UINT (*SKTcpClient - Number Of Digits*) (*$GROUP=User,$CAT=User,$GROUPICON=User.png,$CATICON=User.png*)
	VAR_INPUT
		n : UDINT;
	END_VAR
END_FUNCTION

{REDUND_ERROR} FUNCTION SKTcpClientXor : USINT (*SKTcpClient - Xor*) (*$GROUP=User,$CAT=User,$GROUPICON=User.png,$CATICON=User.png*)
	VAR_INPUT
		in : ARRAY[0..4999] OF USINT;
		len : UINT;
	END_VAR
END_FUNCTION

{REDUND_ERROR} FUNCTION SKTcpClientNewCsvEntry : USINT (*SKTcpClient - New CSV Entries*) (*$GROUP=User,$CAT=User,$GROUPICON=User.png,$CATICON=User.png*)
	VAR_INPUT
		IDstep : STRING[10];
		Description : STRING[100];
		TypeValue : STRING[10];
		MinTol : STRING[10];
		MaxTol : STRING[10];
		Nom : STRING[10];
		MinEle : STRING[10];
		MaxEle : STRING[10];
		Value : STRING[10];
		ValEle : STRING[10];
		Result : STRING[10];
		pData : UDINT;
	END_VAR
END_FUNCTION

{REDUND_ERROR} FUNCTION SKTcpClientNewLoggerEntry : USINT (*SKTcpClient - New Logger Entries*)
	VAR_INPUT
		msg : STRING[1100];
		pData : UDINT;
		entrys : UINT;
	END_VAR
END_FUNCTION

{REDUND_ERROR} FUNCTION SKTcpClientSC : USINT (*SKTcpClient - SC*) (*$GROUP=User,$CAT=User,$GROUPICON=User.png,$CATICON=User.png*)
	VAR_INPUT
		sc : SKTcpClientSC_Type;
	END_VAR
END_FUNCTION
```

#### SKTcpClientTester.c - SKTcpClientTester
```c
/*************************************************************
*
*         projekt: SKTcp - Panasonic
*
*         autor: Ing. Milan Jun
*         company: B+R Automatizace spol. s r.o.
*         date: 10.09.2020
*
*/

#include <bur/plctypes.h>
#ifdef __cplusplus
	extern "C"
	{
#endif
#include "SKTcp.h"
#ifdef __cplusplus
	};
#endif

/* SKTcpClientTester */
void SKTcpClientTester(struct SKTcpClientTester* inst)
{

 if( inst->Enable == 1 ) {

  if(( inst->Cmd.Send == 1 ) && ( inst->Internal.SendOld == 0 )) {
   inst->Internal.cmdSend = 1 ;
  }
  inst->Internal.SendOld = inst->Cmd.Send ;

  if(( inst->Cmd.Close == 1 ) && ( inst->Internal.CloseOld == 0 )) {
   inst->Internal.cmdClose = 1 ;
  } else {
   if( inst->Cmd.Close == 0 ) {
    inst->Internal.cmdClose = 0 ;
   }
  }
  inst->Internal.CloseOld = inst->Cmd.Close ;

  inst->Status.staSending = 0 ;
  inst->Status.staReceiving = 0 ;
  inst->Status.staReadyToSend = 0 ;
  inst->Status.staReadyToClose = 0 ;

  switch( inst->Internal.Step ) {

   case 0:
    inst->Status.staReadyToSend = 1 ;

    if( inst->Internal.cmdSend == 1 ) {
     inst->FBStatus = 0xFFFF ;
     inst->Status.staSent = 0 ;
     inst->Status.staReceived = 0 ;

     inst->Status.staError = 0 ;
     inst->Status.staErrorSent = 0 ;
     inst->Status.staErrorOpen = 0 ;
     inst->Status.staErrorRecv = 0 ;
     inst->Status.staErrorRecvTout = 0 ;
     inst->Status.staErrorOpen = 0 ;
     inst->Status.staErrorIoctl = 0 ;
     inst->Status.staErrorClient = 0 ;
     inst->Status.staErrorConn = 0 ;
     inst->Status.staErrorConnTout = 0 ;

     inst->Status.RecvSize = 0 ;
     memset((void*)&inst->Status.DataRecv[0], 0, sizeof(inst->Status.DataRecv)) ;

     inst->Internal.TimerConn.IN = 1 ;
     inst->Internal.TimerConn.PT = inst->Params.ConnTimeout ;

     inst->Internal.TCP_Open.enable = 1;
     inst->Internal.TCP_Open.pIfAddr = 0;
     inst->Internal.TCP_Open.port = inst->Params.IPportClient;
     inst->Internal.TCP_Open.options = 0;
     TcpOpen(&inst->Internal.TCP_Open);

     if( inst->Internal.TCP_Open.status == 0 ) {
      //inst->Internal.cmdSend = 0 ;
      inst->Internal.Ident = inst->Internal.TCP_Open.ident ;
      inst->Internal.Step = 5;
     }
     else if( inst->Internal.TimerConn.Q == 1 ) {
//      inst->Internal.cmdSend = 0 ;
      inst->Status.staErrorOpen = 1 ;
      inst->Status.staErrorConn = 1 ;
      inst->Status.staErrorConnTout = 1 ;
      inst->Internal.Step = 99;
     } else if( inst->Internal.TCP_Open.status == ERR_FUB_BUSY ) {

     } else {
      if( inst->Internal.TCP_Open.status == tcpERR_ALREADY_EXIST ) {
       inst->Status.staErrorOpen = 1 ;
       inst->Internal.Step = 90;
      } else {
       inst->Status.staErrorOpen = 1 ;
       inst->Internal.Step = 99;
      }
      //inst->Internal.cmdSend = 0 ;
     }
    }

//    else if( inst->Cmd.Close == 1 ) {
//     inst->Cmd.Close = 0 ;
//     inst->Internal.Step = 40 ;
//    }
    break ;

   case 5:
    inst->Internal.linger_opt.lLinger = 0;
    inst->Internal.linger_opt.lOnOff = 1;

    inst->Internal.TCP_Ioctl.enable = 1;
    inst->Internal.TCP_Ioctl.ident = inst->Internal.Ident;
    inst->Internal.TCP_Ioctl.ioctl = tcpSO_LINGER_SET;
    inst->Internal.TCP_Ioctl.pData = (UDINT)&(inst->Internal.linger_opt);
    inst->Internal.TCP_Ioctl.datalen = sizeof(inst->Internal.linger_opt);
    TcpIoctl(&inst->Internal.TCP_Ioctl);

    if( inst->Internal.TCP_Ioctl.status == 0 ) {
     inst->Internal.Step = 10;
    } else if( inst->Internal.TimerConn.Q == 1 ) {
     inst->Status.staErrorOpen = 1 ;
     inst->Status.staErrorConn = 1 ;
     inst->Status.staErrorConnTout = 1 ;
     inst->Internal.Step = 99;
    } else if( inst->Internal.TCP_Ioctl.status == ERR_FUB_BUSY ) {
    } else {
     inst->Status.staErrorIoctl = 1 ;
     inst->Internal.Step = 90;
    }
    break ;

   case 10:
    inst->Internal.TCP_Client.enable = 1;
    inst->Internal.TCP_Client.ident = inst->Internal.Ident ;
    inst->Internal.TCP_Client.portserv = inst->Params.IPportServ ;
    inst->Internal.TCP_Client.pServer = (UDINT)&inst->Params.IPaddrServ[0];
    TcpClient(&inst->Internal.TCP_Client) ;

    if( inst->Internal.TCP_Client.status == 0 ) {
     inst->Internal.Step = 15;
    } else if( inst->Internal.TimerConn.Q == 1 ) {
     inst->Status.staErrorOpen = 1 ;
     inst->Status.staErrorConn = 1 ;
     inst->Status.staErrorConnTout = 1 ;
     inst->Internal.Step = 90;
    } else if( inst->Internal.TCP_Client.status == ERR_FUB_BUSY ) {
    } else if( inst->Internal.TCP_Client.status == tcpERR_INVALID ) {
     inst->Status.staErrorClient = 1 ;
     inst->Status.staErrorConn = 1 ;
     inst->Internal.Step = 90;
    } else {
     inst->Status.staErrorClient = 1 ;
     inst->Internal.Step = 90;
    }
    break ;

   case 15:
    inst->Status.staReadyToSend = 1 ;
    inst->Status.staReadyToClose = 1 ;
    inst->Status.staSending = 0 ;

    if( inst->Cmd.Send == 1 ) {
     inst->Status.RecvSize = 0 ;
     inst->Internal.TimerRecv.IN = 0 ;
     //inst->Internal.cmdSend = 0 ;
     memset((void*)&inst->Status.DataRecv[0], 0, sizeof(inst->Status.DataRecv)) ;
     inst->Internal.Step = 19;
    } else if( inst->Internal.cmdClose == 1 ) {
     inst->Internal.cmdClose = 0 ;
     inst->Internal.Step = 40;
    }
    break ;

   case 19:

    inst->Params.Packet.internal.start = 2;
    inst->Params.Packet.internal.xor = 0;
    inst->Params.Packet.internal.stop = 3;

    if ( inst->Params.Packet.type == 0 || inst->Params.Packet.type == 2 || inst->Params.Packet.type == 3 )
     inst->Params.Packet.internal.length = 3;
    else if ( inst->Params.Packet.type == 1 )
     inst->Params.Packet.internal.length = 34;

    inst->Params.Packet.internal.data_length = inst->Params.Packet.internal.length + SKTcpClientNod(inst->Params.Packet.internal.length);

    memset((UDINT)&(inst->DataSend.send_data_a), 0, sizeof(inst->DataSend.send_data_a));

    inst->DataSend.send_data_a[0] = inst->Params.Packet.internal.data_length;
    inst->DataSend.send_data_a[1] = inst->Params.Packet.type;
    inst->DataSend.send_data_a[2] = inst->Params.Packet.workplace;
    inst->DataSend.send_data_a[3] = inst->Params.Packet.id;

    if (  inst->Params.Packet.type == 1  ) {

     for (inst->Params.Packet.internal.ti = 0; inst->Params.Packet.internal.ti < 32; inst->Params.Packet.internal.ti++)
     {
      inst->DataSend.send_data_a[inst->Params.Packet.internal.ti+4] = inst->Params.Packet.data[inst->Params.Packet.internal.ti];
     }
    }

    // Vypocet XOR
    for (inst->Params.Packet.internal.ti = 0; inst->Params.Packet.internal.ti < inst->Params.Packet.internal.data_length; inst->Params.Packet.internal.ti++)
    {
     inst->Params.Packet.internal.xor = inst->Params.Packet.internal.xor ^ inst->DataSend.send_data_a[inst->Params.Packet.internal.ti];
    }

    memset((UDINT)&(inst->DataSend.DataSend), 0, sizeof(inst->DataSend.DataSend));
    inst->DataSend.DataSend[0] = inst->Params.Packet.internal.start;
    inst->DataSend.DataSend[1] = inst->Params.Packet.internal.data_length;
    inst->DataSend.DataSend[2] = inst->Params.Packet.type;
    inst->DataSend.DataSend[3] = inst->Params.Packet.workplace;
    inst->DataSend.DataSend[4] = inst->Params.Packet.id;
    if (inst->Params.Packet.type == 0 || inst->Params.Packet.type == 2 || inst->Params.Packet.type == 3)
    {
     inst->DataSend.DataSend[5] = inst->Params.Packet.internal.xor;
     inst->DataSend.DataSend[6] = inst->Params.Packet.internal.stop;
    }

    else if (  inst->Params.Packet.type == 1  ) {

     for (inst->Params.Packet.internal.ti = 0; inst->Params.Packet.internal.ti < 32; inst->Params.Packet.internal.ti++)
     {
      inst->DataSend.DataSend[inst->Params.Packet.internal.ti+5] = inst->Params.Packet.data[inst->Params.Packet.internal.ti];

     }
     inst->DataSend.DataSend[37] = inst->Params.Packet.internal.xor;
     inst->DataSend.DataSend[38] = inst->Params.Packet.internal.stop;
    }

	brsmemcpy((UDINT)&(inst->logger.LastDataSend),(UDINT)&inst->DataSend.DataSend, 200);
	//SKTcpClientNewLoggerEntry(inst->logger.LastDataSend, (UDINT)&(inst->logger.SLOGGER), MAX_TRACE_LOGGER_ENTIRES);

    inst->Internal.Step = 20;

    break;

   case 20:

    inst->Status.staSending = 1 ;
    inst->Status.staSent = 0 ;

    inst->Internal.TCP_Send.enable = 1;
    inst->Internal.TCP_Send.ident = inst->Internal.Ident;
    inst->Internal.TCP_Send.pData = (UDINT)&inst->DataSend.DataSend;

    if ( inst->Params.Packet.type == 0 || inst->Params.Packet.type == 2 || inst->Params.Packet.type == 3  )
    {
     inst->Internal.TCP_Send.datalen = inst->Params.Packet.internal.data_length + 3;
    }
    if ( inst->Params.Packet.type == 1  )
    {
     inst->Internal.TCP_Send.datalen = inst->Params.Packet.internal.data_length + 3;
    }

    inst->Internal.TCP_Send.flags = 0;
    TcpSend(&inst->Internal.TCP_Send);

    if( inst->Internal.TCP_Send.status == 0 ) {
     inst->Status.staSent = 1 ;
     if( inst->Params.disRecv == 0 ) {
      inst->Internal.TimerRecv.IN = 0 ;
      inst->Internal.Step = 30;
     }
//     else {
//      if( inst->Params.enaClose == 1 ) {
//       inst->Internal.Step = 40;
//      } else {
//       inst->Internal.Step = 15;
//       inst->Internal.cmdClose = 0 ;
//      }
//     }
    } else if( inst->Internal.TCP_Send.status == ERR_FUB_BUSY )	{
    } else if (( inst->Internal.TCP_Send.status == tcpERR_SENTLEN )
    || ( inst->Internal.TCP_Send.status == tcpERR_NOT_CONNECTED )) {
     inst->Internal.Step = 90;
    } else {
     inst->Status.staErrorSent = 1 ;
     inst->Internal.Step = 90;
    }
    break ;

   case 30:
    inst->Status.staReceiving = 1 ;
    inst->Status.staReceived = 0 ;

    inst->Internal.TimerRecv.IN = 1 ;
    inst->Internal.TimerRecv.PT = inst->Params.RecvTimeout ;

    inst->Internal.TCP_Recv.enable = 1;
    inst->Internal.TCP_Recv.ident = inst->Internal.Ident;
    inst->Internal.TCP_Recv.pData	= (UDINT)&inst->Status.DataRecv[0];
    inst->Internal.TCP_Recv.datamax = sizeof(inst->Status.DataRecv);
    inst->Internal.TCP_Recv.flags = 0;
    TcpRecv(&inst->Internal.TCP_Recv);

    if( inst->Internal.TCP_Recv.status == 0 ) {
     inst->Status.staReceived = 1 ;
     inst->Status.RecvSize = inst->Internal.TCP_Recv.recvlen;
     inst->Status.RecvCounter++ ;

	 brsmemcpy((UDINT)&(inst->logger.LastDataRecv),(UDINT)&inst->Status.DataRecv, 200);
	 //SKTcpClientNewLoggerEntry(inst->logger.LastDataRecv, (UDINT)&(inst->logger.RLOGGER), MAX_TRACE_LOGGER_ENTIRES);

     if( inst->Params.enaClose == 1 ) {
      inst->Internal.Step = 40;
     } else {
      inst->Internal.Step = 15 ;
     }
    } else if( inst->Internal.TCP_Recv.status == tcpERR_NO_DATA ) {
     if( inst->Internal.TimerRecv.Q == 1 ) {
      inst->Status.staErrorRecvTout = 1 ;
      inst->Internal.Step = 90;
     }
    } else if( inst->Internal.TCP_Recv.status == ERR_FUB_BUSY ) {
     if( inst->Internal.TimerRecv.Q == 1 ) {

     }
    } else if( inst->Internal.TCP_Recv.status == tcpERR_NOT_CONNECTED ) {
     inst->Status.staErrorRecv = 1 ;
     inst->Internal.Step = 90;
    } else if( inst->Internal.TimerRecv.Q == 1 ) {
     inst->Status.staErrorRecv = 1 ;
     inst->Internal.TimerRecv.IN = 0 ;
     inst->Internal.Step = 90;
    }
    break ;

   case 40:
    inst->Internal.TCP_Close.enable = 1;
    inst->Internal.TCP_Close.ident = inst->Internal.Ident ;
    inst->Internal.TCP_Close.how = 0;
    TcpClose(&inst->Internal.TCP_Close);

    if( inst->Internal.TCP_Close.status == 0 ) {
     inst->Internal.Ident = 0 ;
     inst->Internal.Step = 100;
     inst->Status.staReceived = 1 ;
    } else if( inst->Internal.TCP_Close.status == ERR_FUB_BUSY ) {
    } else {
     inst->Status.staErrorClose = 1 ;
     inst->Internal.Step = 99;
    }
    break ;

   case 90:
    inst->Internal.TCP_Close.enable = 1;
    inst->Internal.TCP_Close.ident = inst->Internal.Ident;
    inst->Internal.TCP_Close.how = 0;
    TcpClose(&inst->Internal.TCP_Close);

    if( inst->Internal.TCP_Close.status == 0 ) {
     inst->Internal.Ident = 0 ;
     inst->Internal.Step = 99;
    } else if( inst->Internal.TCP_Close.status == ERR_FUB_BUSY ) {
    } else {
     inst->Status.staErrorClose = 1 ;
     inst->Internal.Step = 99;
    }
    break ;

   case 99:
    inst->FBStatus = 1 ;
    inst->Status.staError = 1 ; ;
    inst->Internal.Step = 0;
    inst->Internal.TimerConn.IN = 0 ;
    inst->Internal.cmdSend = 0 ;
    break ;

   case 100:
    inst->FBStatus = 0 ;
    inst->Internal.Step = 0;
    inst->Internal.cmdSend = 0 ;
    inst->Internal.TimerConn.IN = 0 ;
    break ;

  }
 } else {
  if( inst->Cmd.Send == 0 ) {
   inst->FBStatus = 0xFFFE ;
  }

  if( inst->Internal.Ident != 0 ) {
   inst->Internal.TCP_Close.enable = 1;
   inst->Internal.TCP_Close.ident = inst->Internal.Ident;
   inst->Internal.TCP_Close.how = 0;
   TcpClose(&inst->Internal.TCP_Close);

   if( inst->Internal.TCP_Close.status == 0 ) {
    inst->Internal.Ident = 0 ;
   } else if( inst->Internal.TCP_Close.status == ERR_FUB_BUSY ) {
   } else {
   }
  }
  inst->Internal.TimerRecv.IN = 0 ;
  inst->Internal.TimerConn.IN = 0 ;
  inst->Internal.Step = 0 ;
 }

 inst->Internal.EnableOld = inst->Enable ;
 TON(&inst->Internal.TimerRecv) ;
 TON(&inst->Internal.TimerConn) ;

}
```

#### SKTcpClientTrace.c - SKTcpClientTrace
```c
/*************************************************************
*
*         projekt: SKTcp - Panasonic
*
*         autor: Ing. Milan Jun
*         company: B+R Automatizace spol. s r.o.
*         date: 10.09.2020
*
*/

#include <bur/plctypes.h>
#ifdef __cplusplus
	extern "C"
	{
#endif
#include "SKTcp.h"
#ifdef __cplusplus
	};
#endif

/* SKTcpClientTrace */
void SKTcpClientTrace(struct SKTcpClientTrace* inst)
{

 if( inst->Enable == 1 ) {

  if(( inst->Cmd.Send == 1 ) && ( inst->Internal.SendOld == 0 )) {
   inst->Internal.cmdSend = 1 ;
  }
  inst->Internal.SendOld = inst->Cmd.Send ;

  if(( inst->Cmd.Close == 1 ) && ( inst->Internal.CloseOld == 0 )) {
   inst->Internal.cmdClose = 1 ;
  } else {
   if( inst->Cmd.Close == 0 ) {
    inst->Internal.cmdClose = 0 ;
   }
  }
  inst->Internal.CloseOld = inst->Cmd.Close ;

  inst->Status.staSending = 0 ;
  inst->Status.staReceiving = 0 ;
  inst->Status.staReadyToSend = 0 ;
  inst->Status.staReadyToClose = 0 ;

  switch( inst->Internal.Step ) {

   case 0:
    inst->Status.staReadyToSend = 1 ;

    if( inst->Internal.cmdSend == 1 ) {
     inst->FBStatus = 0xFFFF ;
     inst->Status.staSent = 0 ;
     inst->Status.staReceived = 0 ;

     inst->Status.staError = 0 ;
     inst->Status.staErrorSent = 0 ;
     inst->Status.staErrorOpen = 0 ;
     inst->Status.staErrorRecv = 0 ;
     inst->Status.staErrorRecvTout = 0 ;
     inst->Status.staErrorOpen = 0 ;
     inst->Status.staErrorIoctl = 0 ;
     inst->Status.staErrorClient = 0 ;
     inst->Status.staErrorConn = 0 ;
     inst->Status.staErrorConnTout = 0 ;

     inst->Status.RecvSize = 0 ;
     brsmemset((void*)&inst->Status.DataRecv[0], 0, sizeof(inst->Status.DataRecv)) ;

     inst->Internal.TimerConn.IN = 1 ;
     inst->Internal.TimerConn.PT = inst->Params.ConnTimeout ;

     inst->Internal.TCP_Open.enable = 1;
     inst->Internal.TCP_Open.pIfAddr = 0;
     inst->Internal.TCP_Open.port = inst->Params.IPportClient;
     inst->Internal.TCP_Open.options = 0;
     TcpOpen(&inst->Internal.TCP_Open);

     if( inst->Internal.TCP_Open.status == 0 ) {
      //inst->Internal.cmdSend = 0 ;
      inst->Internal.Ident = inst->Internal.TCP_Open.ident ;
      inst->Internal.Step = 5;
     }
     else if( inst->Internal.TimerConn.Q == 1 ) {
      inst->Internal.cmdSend = 0 ;
      inst->Status.staErrorOpen = 1 ;
      inst->Status.staErrorConn = 1 ;
      inst->Status.staErrorConnTout = 1 ;
      inst->Internal.Step = 99;
     } else if( inst->Internal.TCP_Open.status == ERR_FUB_BUSY ) {

     } else {
      if( inst->Internal.TCP_Open.status == tcpERR_ALREADY_EXIST ) {
       inst->Status.staErrorOpen = 1 ;
       inst->Internal.Step = 90;
      } else {
       inst->Status.staErrorOpen = 1 ;
       inst->Internal.Step = 99;
      }
      inst->Internal.cmdSend = 0 ;
     }
    }

    else if( inst->Cmd.Close == 1 ) {
     inst->Cmd.Close = 0 ;
     inst->Internal.Step = 40 ;
    }
    break ;

   case 5:
    inst->Internal.linger_opt.lLinger = 0;
    inst->Internal.linger_opt.lOnOff = 1;

    inst->Internal.TCP_Ioctl.enable = 1;
    inst->Internal.TCP_Ioctl.ident = inst->Internal.Ident;
    inst->Internal.TCP_Ioctl.ioctl = tcpSO_LINGER_SET;
    inst->Internal.TCP_Ioctl.pData = (UDINT)&(inst->Internal.linger_opt);
    inst->Internal.TCP_Ioctl.datalen = sizeof(inst->Internal.linger_opt);
    TcpIoctl(&inst->Internal.TCP_Ioctl);

    if( inst->Internal.TCP_Ioctl.status == 0 ) {
     inst->Internal.Step = 10;
    } else if( inst->Internal.TimerConn.Q == 1 ) {
     inst->Status.staErrorOpen = 1 ;
     inst->Status.staErrorConn = 1 ;
     inst->Status.staErrorConnTout = 1 ;
     inst->Internal.Step = 99;
    } else if( inst->Internal.TCP_Ioctl.status == ERR_FUB_BUSY ) {
    } else {
     inst->Status.staErrorIoctl = 1 ;
     inst->Internal.Step = 90;
    }
    break ;

   case 10:
    inst->Internal.TCP_Client.enable = 1;
    inst->Internal.TCP_Client.ident = inst->Internal.Ident ;
    inst->Internal.TCP_Client.portserv = inst->Params.IPportServ ;
    inst->Internal.TCP_Client.pServer = (UDINT)&inst->Params.IPaddrServ[0];
    TcpClient(&inst->Internal.TCP_Client) ;

    if( inst->Internal.TCP_Client.status == 0 ) {
     inst->Internal.Step = 15;
    } else if( inst->Internal.TimerConn.Q == 1 ) {
     inst->Status.staErrorOpen = 1 ;
     inst->Status.staErrorConn = 1 ;
     inst->Status.staErrorConnTout = 1 ;
     inst->Internal.Step = 90;
    } else if( inst->Internal.TCP_Client.status == ERR_FUB_BUSY ) {
    } else if( inst->Internal.TCP_Client.status == tcpERR_INVALID ) {
     inst->Status.staErrorClient = 1 ;
     inst->Status.staErrorConn = 1 ;
     inst->Internal.Step = 90;
    } else {
     inst->Status.staErrorClient = 1 ;
     inst->Internal.Step = 90;
    }
    break ;

   case 15:
    inst->Status.staReadyToSend = 1 ;
    //inst->Status.staReadyToClose = 1 ;
    inst->Status.staSending = 0 ;

    if ( inst->Internal.cmdSend == 1 ) {
     inst->Status.RecvSize = 0 ;
     inst->Internal.TimerRecv.IN = 0 ;
     inst->Internal.cmdSend = 0 ;
     brsmemset((void*)&inst->Status.DataRecv, 0, sizeof(inst->Status.DataRecv)) ;

     brsmemset((void*)&inst->Internal.Splitter.out, 0, sizeof(inst->Internal.Splitter.out));
     inst->Internal.Step = 18;
    }
    //else if( inst->Internal.cmdClose == 1 ) {
    // inst->Internal.cmdClose = 0 ;
    // inst->Internal.Step = 40;
    //}
    break ;

			case 18:

   	inst->Internal.oneskorenie.IN = 1;
				inst->Internal.oneskorenie.PT = 1000; //ms

				if ( inst->Internal.oneskorenie.Q == 1 ) {
					inst->Internal.oneskorenie.IN = 0;
					inst->Internal.Step = 19;
				}

				TON(&inst->Internal.oneskorenie);

    break ;

   case 19:

    inst->Params.Packet.internal.start = 0x02;
    inst->Params.Packet.internal.length_int = 0;
    //inst->Params.Packet.internal.xor = 0;
    inst->Params.Packet.internal.stop = 0x03;

    brsmemset((UDINT)&(inst->Params.Packet.internal.length_str), 0, sizeof(inst->Params.Packet.internal.length_str));
    brsmemset((UDINT)&(inst->Params.Packet.internal.xor_str), 0, sizeof(inst->Params.Packet.internal.xor_str));

    brsmemset((UDINT)&(inst->DataSend.send_data_a), 0, sizeof(inst->DataSend.send_data_a));
    brsstrcat((UDINT)&(inst->DataSend.send_data_a), (UDINT)&(inst->Params.Packet.type));
    brsstrcat((UDINT)&(inst->DataSend.send_data_a), (UDINT)&("|"));
    brsstrcat((UDINT)&(inst->DataSend.send_data_a), (UDINT)&(inst->Params.Packet.workplace));
    brsstrcat((UDINT)&(inst->DataSend.send_data_a), (UDINT)&("|"));
    brsstrcat((UDINT)&(inst->DataSend.send_data_a), (UDINT)&(inst->Params.Packet.rfid));
    brsstrcat((UDINT)&(inst->DataSend.send_data_a), (UDINT)&("|"));
    brsstrcat((UDINT)&(inst->DataSend.send_data_a), (UDINT)&(inst->Params.Packet.master));
    brsstrcat((UDINT)&(inst->DataSend.send_data_a), (UDINT)&("|"));
    brsstrcat((UDINT)&(inst->DataSend.send_data_a), (UDINT)&(inst->Params.Packet.dps1));
    brsstrcat((UDINT)&(inst->DataSend.send_data_a), (UDINT)&("|"));
    brsstrcat((UDINT)&(inst->DataSend.send_data_a), (UDINT)&(inst->Params.Packet.dps2));
    brsstrcat((UDINT)&(inst->DataSend.send_data_a), (UDINT)&("|"));
    brsstrcat((UDINT)&(inst->DataSend.send_data_a), (UDINT)&(inst->Params.Packet.dps3));
    brsstrcat((UDINT)&(inst->DataSend.send_data_a), (UDINT)&("|"));
    brsstrcat((UDINT)&(inst->DataSend.send_data_a), (UDINT)&(inst->Params.Packet.dps4));
    brsstrcat((UDINT)&(inst->DataSend.send_data_a), (UDINT)&("|"));
    brsstrcat((UDINT)&(inst->DataSend.send_data_a), (UDINT)&(inst->Params.Packet.dps5));
    brsstrcat((UDINT)&(inst->DataSend.send_data_a), (UDINT)&("|"));
    brsstrcat((UDINT)&(inst->DataSend.send_data_a), (UDINT)&(inst->Params.Packet.operator_id));
    brsstrcat((UDINT)&(inst->DataSend.send_data_a), (UDINT)&("|"));
    brsstrcat((UDINT)&(inst->DataSend.send_data_a), (UDINT)&(inst->Params.Packet.data_report));
    brsstrcat((UDINT)&(inst->DataSend.send_data_a), (UDINT)&("|"));
    brsstrcat((UDINT)&(inst->DataSend.send_data_a), (UDINT)&(inst->Params.Packet.result));

    inst->Params.Packet.internal.length_int = brsstrlen((UDINT)&inst->DataSend.send_data_a);
    inst->Params.Packet.internal.length_int = inst->Params.Packet.internal.length_int + SKTcpClientNod(inst->Params.Packet.internal.length_int);

    brsitoa(inst->Params.Packet.internal.length_int,(UDINT)&(inst->Params.Packet.internal.length_str));

    brsmemset((UDINT)&(inst->DataSend.send_data_b), 0, sizeof(inst->DataSend.send_data_b));
    brsstrcat((UDINT)&(inst->DataSend.send_data_b), (UDINT)&(inst->Params.Packet.internal.length_str));
    brsstrcat((UDINT)&(inst->DataSend.send_data_b), (UDINT)&("|"));
    brsstrcat((UDINT)&(inst->DataSend.send_data_b), (UDINT)&(inst->Params.Packet.type));
    brsstrcat((UDINT)&(inst->DataSend.send_data_b), (UDINT)&("|"));
    brsstrcat((UDINT)&(inst->DataSend.send_data_b), (UDINT)&(inst->Params.Packet.workplace));
    brsstrcat((UDINT)&(inst->DataSend.send_data_b), (UDINT)&("|"));
    brsstrcat((UDINT)&(inst->DataSend.send_data_b), (UDINT)&(inst->Params.Packet.rfid));
    brsstrcat((UDINT)&(inst->DataSend.send_data_b), (UDINT)&("|"));
    brsstrcat((UDINT)&(inst->DataSend.send_data_b), (UDINT)&(inst->Params.Packet.master));
    brsstrcat((UDINT)&(inst->DataSend.send_data_b), (UDINT)&("|"));
    brsstrcat((UDINT)&(inst->DataSend.send_data_b), (UDINT)&(inst->Params.Packet.dps1));
    brsstrcat((UDINT)&(inst->DataSend.send_data_b), (UDINT)&("|"));
    brsstrcat((UDINT)&(inst->DataSend.send_data_b), (UDINT)&(inst->Params.Packet.dps2));
    brsstrcat((UDINT)&(inst->DataSend.send_data_b), (UDINT)&("|"));
    brsstrcat((UDINT)&(inst->DataSend.send_data_b), (UDINT)&(inst->Params.Packet.dps3));
    brsstrcat((UDINT)&(inst->DataSend.send_data_b), (UDINT)&("|"));
    brsstrcat((UDINT)&(inst->DataSend.send_data_b), (UDINT)&(inst->Params.Packet.dps4));
    brsstrcat((UDINT)&(inst->DataSend.send_data_b), (UDINT)&("|"));
    brsstrcat((UDINT)&(inst->DataSend.send_data_b), (UDINT)&(inst->Params.Packet.dps5));
    brsstrcat((UDINT)&(inst->DataSend.send_data_b), (UDINT)&("|"));
    brsstrcat((UDINT)&(inst->DataSend.send_data_b), (UDINT)&(inst->Params.Packet.operator_id));
    brsstrcat((UDINT)&(inst->DataSend.send_data_b), (UDINT)&("|"));
    brsstrcat((UDINT)&(inst->DataSend.send_data_b), (UDINT)&(inst->Params.Packet.data_report));
    brsstrcat((UDINT)&(inst->DataSend.send_data_b), (UDINT)&("|"));
    brsstrcat((UDINT)&(inst->DataSend.send_data_b), (UDINT)&(inst->Params.Packet.result));
    brsstrcat((UDINT)&(inst->DataSend.send_data_b), (UDINT)&("|"));

    inst->Params.Packet.internal.xor_str = SKTcpClientXor(inst->DataSend.send_data_b,inst->Params.Packet.internal.length_int+3);

    brsmemset((UDINT)&(inst->DataSend.DataSend), 0, sizeof(inst->DataSend.DataSend));
    inst->DataSend.DataSend[0] = inst->Params.Packet.internal.start;
    brsstrcat((UDINT)&(inst->DataSend.DataSend), (UDINT)&(inst->Params.Packet.internal.length_str));
    brsstrcat((UDINT)&(inst->DataSend.DataSend), (UDINT)&("|"));
    brsstrcat((UDINT)&(inst->DataSend.DataSend), (UDINT)&(inst->Params.Packet.type));
    brsstrcat((UDINT)&(inst->DataSend.DataSend), (UDINT)&("|"));
    brsstrcat((UDINT)&(inst->DataSend.DataSend), (UDINT)&(inst->Params.Packet.workplace));
    brsstrcat((UDINT)&(inst->DataSend.DataSend), (UDINT)&("|"));
    brsstrcat((UDINT)&(inst->DataSend.DataSend), (UDINT)&(inst->Params.Packet.rfid));
    brsstrcat((UDINT)&(inst->DataSend.DataSend), (UDINT)&("|"));
    brsstrcat((UDINT)&(inst->DataSend.DataSend), (UDINT)&(inst->Params.Packet.master));
    brsstrcat((UDINT)&(inst->DataSend.DataSend), (UDINT)&("|"));
    brsstrcat((UDINT)&(inst->DataSend.DataSend), (UDINT)&(inst->Params.Packet.dps1));
    brsstrcat((UDINT)&(inst->DataSend.DataSend), (UDINT)&("|"));
    brsstrcat((UDINT)&(inst->DataSend.DataSend), (UDINT)&(inst->Params.Packet.dps2));
    brsstrcat((UDINT)&(inst->DataSend.DataSend), (UDINT)&("|"));
    brsstrcat((UDINT)&(inst->DataSend.DataSend), (UDINT)&(inst->Params.Packet.dps3));
    brsstrcat((UDINT)&(inst->DataSend.DataSend), (UDINT)&("|"));
    brsstrcat((UDINT)&(inst->DataSend.DataSend), (UDINT)&(inst->Params.Packet.dps4));
    brsstrcat((UDINT)&(inst->DataSend.DataSend), (UDINT)&("|"));
    brsstrcat((UDINT)&(inst->DataSend.DataSend), (UDINT)&(inst->Params.Packet.dps5));
    brsstrcat((UDINT)&(inst->DataSend.DataSend), (UDINT)&("|"));
    brsstrcat((UDINT)&(inst->DataSend.DataSend), (UDINT)&(inst->Params.Packet.operator_id));
    brsstrcat((UDINT)&(inst->DataSend.DataSend), (UDINT)&("|"));
    brsstrcat((UDINT)&(inst->DataSend.DataSend), (UDINT)&(inst->Params.Packet.data_report));
    brsstrcat((UDINT)&(inst->DataSend.DataSend), (UDINT)&("|"));
    brsstrcat((UDINT)&(inst->DataSend.DataSend), (UDINT)&(inst->Params.Packet.result));
    brsstrcat((UDINT)&(inst->DataSend.DataSend), (UDINT)&("|"));

	inst->Params.Packet.internal.ret_len = strlen((UDINT)&inst->DataSend.DataSend);

	if ( inst->Params.Packet.internal.xor_str != 0 )
     brsstrcat((UDINT)&(inst->DataSend.DataSend), (UDINT)&(inst->Params.Packet.internal.xor_str));
    else{
	 inst->DataSend.DataSend[inst->Params.Packet.internal.ret_len] = 0x00;
	 inst->DataSend.DataSend[inst->Params.Packet.internal.ret_len+1] = 0x03;
    }

    brsmemcpy((UDINT)&(inst->logger.LastDataSend),(UDINT)&inst->DataSend.DataSend, 5000);
    //SKTcpClientNewLoggerEntry(inst->logger.LastDataSend, (UDINT)&(inst->logger.SLOGGER), MAX_TRACE_LOGGER_ENTIRES);

    inst->Internal.Step = 20;

   case 20:

    inst->Status.staSending = 1 ;
    inst->Status.staSent = 0 ;

    inst->Internal.Splitter.enable = 0;

    inst->Internal.TCP_Send.enable = 1;
    inst->Internal.TCP_Send.ident = inst->Internal.Ident;
    inst->Internal.TCP_Send.pData = (UDINT)&inst->DataSend.DataSend;
    inst->Internal.TCP_Send.datalen = sizeof(inst->DataSend.DataSend);
    inst->Internal.TCP_Send.flags = 0;
    TcpSend(&inst->Internal.TCP_Send);

    if( inst->Internal.TCP_Send.status == 0 ) {
     inst->Status.staSent = 1 ;
     if( inst->Params.disRecv == 0 ) {
      inst->Internal.TimerRecv.IN = 0 ;
      inst->Internal.Step = 30;
     }
//     else {
//      if( inst->Params.enaClose == 1 ) {
//       inst->Internal.Step = 40;
//      }
//      else {
//       inst->Internal.Step = 15;
//       inst->Internal.cmdClose = 0 ;
//      }
//     }
    } else if( inst->Internal.TCP_Send.status == ERR_FUB_BUSY )	{
    } else if (( inst->Internal.TCP_Send.status == tcpERR_SENTLEN ) || ( inst->Internal.TCP_Send.status == tcpERR_NOT_CONNECTED )) {
     inst->Internal.Step = 90;
    } else {
     inst->Status.staErrorSent = 1 ;
     inst->Internal.Step = 90;
    }
    break;

   case 30:

    inst->Status.staReceiving = 1 ;
    inst->Status.staReceived = 0 ;

    inst->Internal.TimerRecv.IN = 1 ;
    inst->Internal.TimerRecv.PT = inst->Params.RecvTimeout ;

    inst->Internal.TCP_Recv.enable = 1;
    inst->Internal.TCP_Recv.ident = inst->Internal.Ident;
    inst->Internal.TCP_Recv.pData	= (UDINT)&inst->Status.DataRecv;
    inst->Internal.TCP_Recv.datamax = sizeof(inst->Status.DataRecv);
    inst->Internal.TCP_Recv.flags = 0;
    TcpRecv(&inst->Internal.TCP_Recv);

    if( inst->Internal.TCP_Recv.status == 0 ) {
     inst->Status.staReceived = 1 ;
     inst->Status.RecvSize = inst->Internal.TCP_Recv.recvlen;
     inst->Status.RecvCounter++ ;

 	 brsmemcpy((UDINT)&(inst->logger.LastDataRecv),(UDINT)&inst->Status.DataRecv, 5000);
     //SKTcpClientNewLoggerEntry(inst->logger.LastDataRecv, (UDINT)&(inst->logger.RLOGGER), MAX_TRACE_LOGGER_ENTIRES);

     brsmemcpy((UDINT)&inst->Internal.Splitter.iSelector,(UDINT)&("|"),sizeof("|"));
     brsmemcpy((UDINT)&inst->Internal.Splitter.iInputString,(UDINT)&(inst->Status.DataRecv),sizeof(inst->Status.DataRecv));
     inst->Internal.Splitter.enable = 1;
     inst->Internal.Step = 40;

     if( inst->Params.enaClose == 1 ) {
      inst->Internal.Step = 40;
     } else {
      inst->Internal.Step = 15;
     }
    } else if( inst->Internal.TCP_Recv.status == tcpERR_NO_DATA ) {
     if( inst->Internal.TimerRecv.Q == 1 ) {
      inst->Status.staErrorRecvTout = 1 ;
      inst->Internal.Step = 90;
     }
    } else if( inst->Internal.TCP_Recv.status == ERR_FUB_BUSY ) {
     if( inst->Internal.TimerRecv.Q == 1 ) {

     }
    } else if( inst->Internal.TCP_Recv.status == tcpERR_NOT_CONNECTED ) {
     inst->Status.staErrorRecv = 1 ;
     inst->Internal.Step = 90;
    } else if( inst->Internal.TimerRecv.Q == 1 ) {
     inst->Status.staErrorRecv = 1 ;
     inst->Internal.TimerRecv.IN = 0 ;
     inst->Internal.Step = 90;
    }
    break ;

   case 40:
    inst->Internal.TCP_Close.enable = 1;
    inst->Internal.TCP_Close.ident = inst->Internal.Ident ;
    inst->Internal.TCP_Close.how = 0;
    TcpClose(&inst->Internal.TCP_Close);

    if( inst->Internal.TCP_Close.status == 0 ) {
     inst->Internal.Ident = 0 ;
     inst->Internal.Step = 100;
     inst->Status.staReceived = 1 ;
    } else if( inst->Internal.TCP_Close.status == ERR_FUB_BUSY ) {
    } else {
     inst->Status.staErrorClose = 1 ;
     inst->Internal.Step = 99;
    }
    break ;

   case 90:
    inst->Internal.TCP_Close.enable = 1;
    inst->Internal.TCP_Close.ident = inst->Internal.Ident;
    inst->Internal.TCP_Close.how = 0;
    TcpClose(&inst->Internal.TCP_Close);

    if( inst->Internal.TCP_Close.status == 0 ) {
     inst->Internal.Ident = 0 ;
     inst->Internal.Step = 99;
    } else if( inst->Internal.TCP_Close.status == ERR_FUB_BUSY ) {
    } else {
     inst->Status.staErrorClose = 1 ;
     inst->Internal.Step = 99;
    }
    break ;

   case 99:
    inst->FBStatus = 1 ;
    inst->Status.staError = 1 ; ;
    inst->Internal.Step = 0;
    inst->Internal.TimerConn.IN = 0 ;
    inst->Internal.cmdSend = 0 ;
    break ;

   case 100:
    inst->FBStatus = 0 ;
    inst->Internal.Step = 0;
    inst->Internal.cmdSend = 0 ;
    inst->Internal.TimerConn.IN = 0 ;
    break ;

  }
 } else {
  if( inst->Cmd.Send == 0 ) {
   inst->FBStatus = 0xFFFE ;
  }

  if( inst->Internal.Ident != 0 ) {
   inst->Internal.TCP_Close.enable = 1;
   inst->Internal.TCP_Close.ident = inst->Internal.Ident;
   inst->Internal.TCP_Close.how = 0;
   TcpClose(&inst->Internal.TCP_Close);

   if( inst->Internal.TCP_Close.status == 0 ) {
    inst->Internal.Ident = 0 ;
   } else if( inst->Internal.TCP_Close.status == ERR_FUB_BUSY ) {
   } else {
   }
  }
  inst->Internal.TimerRecv.IN = 0 ;
  inst->Internal.TimerConn.IN = 0 ;
  inst->Internal.Step = 0 ;
 }

 inst->Internal.EnableOld = inst->Enable ;
 TON(&inst->Internal.TimerRecv) ;
 TON(&inst->Internal.TimerConn) ;
 SKTcpClientSplitter(&inst->Internal.Splitter);

}
```

#### SKTcpClientSplitter.c - SKTcpClientSplitter
```c
/*************************************************************
*
*         projekt: SKTcp - Panasonic
*
*         autor: Ing. Milan Jun
*         company: B+R Automatizace spol. s r.o.
*         date: 10.09.2020
*
*/

#include <bur/plctypes.h>
#ifdef __cplusplus
	extern "C"
	{
#endif
	#include "SKTcp.h"
#ifdef __cplusplus
	};
#endif

/* SKTcpClientSplitter */
void SKTcpClientSplitter(struct SKTcpClientSplitter* inst)
{

 if ( inst->enable == 0 )
 {

  inst->done = 0;

  brsmemset((UDINT)&(inst->out), 0, sizeof(inst->out));
  brsmemset((UDINT)&(inst->OUT_Master), 0, sizeof(inst->OUT_Master));
  brsmemset((UDINT)&(inst->OUT_Typ), 0, sizeof(inst->OUT_Typ));
  brsmemset((UDINT)&(inst->OUT_Result), 0, sizeof(inst->OUT_Result));
  brsmemset((UDINT)&(inst->tmpInputString), 0, sizeof(inst->tmpInputString));
  brsmemset((UDINT)&(inst->tmpString), 0, sizeof(inst->tmpString));
  brsmemset((UDINT)&(inst->idx), 0, sizeof(inst->idx));

 }
 else if ( inst->enable == 1 )
 {

  if ( inst->enable == 1 && inst->enableOld==0 )
  {
   inst->enableOld = 1;

   brsmemcpy ((UDINT)&(inst->tmpInputString),(UDINT)&(inst->iInputString), brsstrlen((UDINT)&(inst->iInputString)));

   inst->idx[1] = 0;

   if ( strlen((UDINT)&(inst->iInputString)) != 0 )
   {

    for (inst->idx[0] = 0; inst->idx[0] < brsstrlen(inst->iInputString) ; inst->idx[0]++)
    {

     if ( inst->iSelector != inst->tmpInputString[inst->idx[0]] )
     {
      brsmemcpy((UDINT)&(inst->tmpString),(UDINT)&(inst->tmpInputString[inst->idx[0]]),1);
      brsstrcat((UDINT)&(inst->out[inst->idx[1]]),(UDINT)&(inst->tmpString));

     }
     else
     {
      inst->idx[1]++;
     }

    }
	brsmemcpy((UDINT)&(inst->OUT_Master),(UDINT)&(inst->out[4]),30);
		brsmemcpy((UDINT)&(inst->OUT_Typ),(UDINT)&(inst->out[1]),1);
		brsmemcpy((UDINT)&(inst->OUT_Result),(UDINT)&(inst->out[12]),2);
   }

  }

 }

 inst->enableOld = inst->enable;

}
```

#### SKTcpClientXor.c - SKTcpClientXor
```c
/*************************************************************
*
*         projekt: SKTcp - Panasonic
*
*         autor: Ing. Milan Jun
*         company: B+R Automatizace spol. s r.o.
*         date: 10.09.2020
*
*/

#include <bur/plctypes.h>
#ifdef __cplusplus
	extern "C"
	{
#endif
	#include "SKTcp.h"
#ifdef __cplusplus
	};
#endif

/* SKTcpClientXor */
unsigned char SKTcpClientXor(unsigned char in[4999], unsigned short len)
{

 unsigned char xor_byte = 0;
 unsigned int tI = 0;

 for (tI = 0; tI < len; tI++) xor_byte = xor_byte ^ in[tI];

 return xor_byte;

}
```

#### SKTcpClientNod.c - SKTcpClientNod
```c
/*************************************************************
*
*         projekt: SKTcp - Panasonic
*
*         autor: Ing. Milan Jun
*         company: B+R Automatizace spol. s r.o.
*         date: 10.09.2020
*
*/

#include <bur/plctypes.h>
#ifdef __cplusplus
	extern "C"
	{
#endif
	#include "SKTcp.h"
#ifdef __cplusplus
	};
#endif

/* SKTcpClientNod */
unsigned short SKTcpClientNod(unsigned long n)
{

 unsigned int count = 0;

 while (n != 0) { n /= 10; ++count; }

 return count;

}
```

#### SKTcpClientEdge.c - SKTcpClientEdge
```c
/*************************************************************
*
*         projekt: SKTcp - Panasonic
*
*         autor: Ing. Milan Jun
*         company: B+R Automatizace spol. s r.o.
*         date: 10.09.2020
*
*/

#include <bur/plctypes.h>
#ifdef __cplusplus
	extern "C"
	{
#endif
	#include "SKTcp.h"
#ifdef __cplusplus
	};
#endif

/* SKTcpClientEdge */
void SKTcpClientEdge(struct SKTcpClientEdge* inst)
{

 inst->Q = ( ! inst->CLK == inst->Last_State) ;

 inst->Last_State = inst->CLK;

}
```

#### SKTcpClientNewCsvEntry.c - SKTcpClientNewCsvEntry
```c
/*************************************************************
*
*         projekt: SKTcp - Panasonic
*
*         autor: Ing. Milan Jun
*         company: B+R Automatizace spol. s r.o.
*         date: 21.09.2020
*
*/

#include <bur/plctypes.h>
#ifdef __cplusplus
	extern "C"
	{
#endif
	#include "SKTcp.h"
#ifdef __cplusplus
	};
#endif

/* SKTcpClientNewCsvEntry */
unsigned char SKTcpClientNewCsvEntry(plcstring* IDstep, plcstring* Description, plcstring* TypeValue, plcstring* MinTol, plcstring* MaxTol, plcstring* Nom, plcstring* MinEle, plcstring* MaxEle, plcstring* Value, plcstring* ValEle, plcstring* Result, unsigned long pData)
{

	/* SKTcpClientNewCsvEntry('IDstep','Description','TypeValue','MinTol','MaxTol','Nom','MinEle','MaxEle','Value','ValEle','Result', ADR(CSV)); */

	brsstrcat((void*)pData, IDstep);
	brsstrcat((void*)pData, (UDINT)&";");
	brsstrcat((void*)pData, Description);
	brsstrcat((void*)pData, (UDINT)&";");
	brsstrcat((void*)pData, TypeValue);
	brsstrcat((void*)pData, (UDINT)&";");
	brsstrcat((void*)pData, MinTol);
	brsstrcat((void*)pData, (UDINT)&";");
	brsstrcat((void*)pData, MaxTol);
	brsstrcat((void*)pData, (UDINT)&";");
	brsstrcat((void*)pData, Nom);
	brsstrcat((void*)pData, (UDINT)&";");
	brsstrcat((void*)pData, MinEle);
	brsstrcat((void*)pData, (UDINT)&";");
	brsstrcat((void*)pData, MaxEle);
	brsstrcat((void*)pData, (UDINT)&";");
	brsstrcat((void*)pData, Value);
	brsstrcat((void*)pData, (UDINT)&";");
	brsstrcat((void*)pData, ValEle);
	brsstrcat((void*)pData, (UDINT)&";");
	brsstrcat((void*)pData, Result);
	brsstrcat((void*)pData, (UDINT)&("\r"));

	return 0;
}
```

#### SKTcpClientNewLoggerEntry.c - SKTcpClientNewLoggerEntry
```c
/*************************************************************
*
*         projekt: SKTcp - Panasonic
*
*         autor: Ing. Milan Jun
*         company: B+R Automatizace spol. s r.o.
*         date: 21.09.2020
*
*/

#include <bur/plctypes.h>
#ifdef __cplusplus
	extern "C"
	{
#endif
	#include "SKTcp.h"
#ifdef __cplusplus
	};
#endif

/* SKTcpClientNewLoggerEntry */
unsigned char SKTcpClientNewLoggerEntry(plcstring* msg, UDINT pData, UINT entrys)
{

	RTCtime_typ	RTCtime_struct;
	STRING lstr1[5000], lstr2[5000];

	if ((entrys > 0) && (pData != 0))
	{
		brsstrcpy(lstr1, "");
		brsstrcpy(lstr2, "");
		RTC_gettime(&RTCtime_struct);
		brsitoa(RTCtime_struct.hour, (UDINT)&lstr1);
		if(brsstrlen(lstr1) == 1) brsstrcat(lstr2, "0");
		brsstrcat(lstr2, lstr1);
		brsstrcat(lstr2, ":");
		brsitoa(RTCtime_struct.minute, (UDINT)&lstr1);
		if(brsstrlen(lstr1) == 1) brsstrcat(lstr2, "0");
		brsstrcat(lstr2, lstr1);
		brsstrcat(lstr2, ":");
		brsitoa(RTCtime_struct.second, (UDINT)&lstr1);
		if(brsstrlen(lstr1) == 1) brsstrcat(lstr2, "0");
		brsstrcat(lstr2, lstr1);
		brsstrcat(lstr2, ":");
		brsitoa(RTCtime_struct.millisec, (UDINT)&lstr1);
		if(brsstrlen(lstr1) == 1) brsstrcat(lstr2, "00");
		if(brsstrlen(lstr1) == 2) brsstrcat(lstr2, "0");
		brsstrcat(lstr2, lstr1);
		brsstrcat(lstr2, " ");
		brsstrcat(lstr2, msg);
		brsmemmove((void*)(pData)+5001, (void*)pData, 5001*(entrys-1));
		brsstrcpy((void*)pData, lstr2);
	}

	return 0;

}
```

#### SKTcpClientFTP.c - SKTcpClientFTP
```c
/*************************************************************
*
*         projekt: SKTcp - Panasonic
*
*         autor: Ing. Milan Jun
*         company: B+R Automatizace spol. s r.o.
*         date: 21.09.2020
*
*/

#include <bur/plctypes.h>
#ifdef __cplusplus
extern "C"
{
#endif
#include "SKTcp.h"
#ifdef __cplusplus
};
#endif

/* SKTcpClientFTP */
void SKTcpClientFTP(struct SKTcpClientFTP* inst)
{

if ( inst->enable == 1 ) {

	inst->active = 1;

	SKTcpClientSC(&inst->internal.sc);

	switch (inst->internal.sc.step)
	{

		case 0:

			if ( inst->send == 1 ) {
					inst->internal.sc.bNext = 1;
			}

			break;

		case 1:

			brsstrcpy((UDINT)&inst->internal.sc.StepName,(UDINT)&("DevLink - source"));

			if ( inst->internal.sc.edge == 0 ){
				inst->internal.fb.Devlink_0.enable = 1;
				inst->internal.fb.Devlink_0.pDevice = inst->param.src.pDevice;
				inst->internal.fb.Devlink_0.pParam = inst->param.src.pParam;
				inst->internal.sc.edge = 1;
			}

			DevLink(&inst->internal.fb.Devlink_0);

			if (inst->internal.fb.Devlink_0.status == ERR_OK)
			{
				inst->internal.src_handle = inst->internal.fb.Devlink_0.handle;
				inst->internal.sc.bNext = 1;
			}
			else if ( inst->internal.fb.Devlink_0.status == ERR_FUB_BUSY )
			{

			}
   else if ( inst->internal.fb.Devlink_0.status == fiERR_DEVICE_ALREADY_EXIST ) {
    inst->internal.sc.bJump = 1;
    inst->internal.sc.step = 6;
    }
			break;

		case 2:

			brsstrcpy((UDINT)&inst->internal.sc.StepName,(UDINT)&("DevLink - destination"));

			inst->internal.fb.Devlink_0.enable = 1;
			inst->internal.fb.Devlink_0.pDevice = inst->param.dest.pDevice;
			inst->internal.fb.Devlink_0.pParam = inst->param.dest.pParam;

			DevLink(&inst->internal.fb.Devlink_0);

			if (inst->internal.fb.Devlink_0.status == ERR_OK)
			{
				inst->internal.dest_handle = inst->internal.fb.Devlink_0.handle;
				inst->internal.sc.bNext = 1;
			}
			else if ( inst->internal.fb.Devlink_0.status == ERR_FUB_BUSY )
			{

			}
    else if ( inst->internal.fb.Devlink_0.status == fiERR_DEVICE_ALREADY_EXIST ) {
     inst->internal.sc.bJump = 1;
     inst->internal.sc.step = 6;
    }
			break;

		case 3:

			brsstrcpy((UDINT)&inst->internal.sc.StepName,(UDINT)&("DirInfo"));

			inst->internal.fb.DirInfo_0.enable = 1;
			inst->internal.fb.DirInfo_0.pDevice = inst->param.src.pDevice;
			inst->internal.fb.DirInfo_0.pPath = inst->param.src.pPath;

			DirInfo(&inst->internal.fb.DirInfo_0);

			if (inst->internal.fb.DirInfo_0.filenum == 1 && inst->internal.fb.DirInfo_0.status == ERR_OK )
			{
				inst->internal.sc.bNext = 1;
			}
			else if ( inst->internal.fb.DirInfo_0.status == ERR_FUB_BUSY )
			{

			}
			break;

		case 4:

			brsstrcpy((UDINT)&inst->internal.sc.StepName,(UDINT)&("DirRead"));

			inst->internal.fb.DirRead_0.enable = 1;
			inst->internal.fb.DirRead_0.pDevice = inst->param.src.pDevice;
			inst->internal.fb.DirRead_0.pPath = inst->param.src.pPath;
			inst->internal.fb.DirRead_0.option = fiFILE;
			inst->internal.fb.DirRead_0.pData = (UDINT)&inst->status.src.pData;
			inst->internal.fb.DirRead_0.data_len = sizeof(fiDIR_READ_DATA);

			DirRead(&inst->internal.fb.DirRead_0);

			if (inst->internal.fb.DirRead_0.status == ERR_OK)
			{
				inst->internal.sc.bNext = 1;
			}
			else if ( inst->internal.fb.DirRead_0.status == ERR_FUB_BUSY )
			{

			}
			break;

		case 5:

			brsstrcpy((UDINT)&inst->internal.sc.StepName,(UDINT)&("FileCopy"));

			inst->internal.fb.FileCopy_0.enable = 1;
			inst->internal.fb.FileCopy_0.pSrcDev = inst->param.src.pDevice;
			inst->internal.fb.FileCopy_0.pSrc = inst->status.src.pData.Filename;
			inst->internal.fb.FileCopy_0.pDestDev = inst->param.dest.pDevice;
			inst->internal.fb.FileCopy_0.pDest = inst->param.dest.pNewName;
            inst->internal.fb.FileCopy_0.option = fiOVERWRITE;

			FileCopy(&inst->internal.fb.FileCopy_0);

			if (inst->internal.fb.FileCopy_0.status == ERR_OK )
			{
				inst->internal.sc.bNext = 1;
			}
			else if ( inst->internal.fb.FileCopy_0.status == ERR_FUB_BUSY )
			{

			}
			break;

		case 6:

			brsstrcpy((UDINT)&inst->internal.sc.StepName,(UDINT)&("File Delete"));

			inst->internal.fb.FileDelete_0.enable = 1;
			inst->internal.fb.FileDelete_0.pDevice = inst->param.src.pDevice;
			inst->internal.fb.FileDelete_0.pName = (UDINT)&inst->status.src.pData.Filename;

			FileDelete(&inst->internal.fb.FileDelete_0);

			if (inst->internal.fb.FileDelete_0.status == ERR_OK)
			{
				inst->internal.sc.bNext = 1;
			}
    else if ( inst->internal.fb.FileDelete_0.status == ERR_FUB_BUSY )
    {

    }
			break;

		case 7:

			brsstrcpy((UDINT)&inst->internal.sc.StepName,(UDINT)&("DevUnlink - source"));

			inst->internal.fb.DevUnlink_0.enable = 1;
			inst->internal.fb.DevUnlink_0.handle = inst->internal.src_handle;

			DevUnlink(&inst->internal.fb.DevUnlink_0);

			if (inst->internal.fb.DevUnlink_0.status == ERR_OK)
			{
				inst->internal.fb.DevUnlink_0.enable = 0;
				inst->internal.src_handle = 0;
				inst->internal.sc.bNext = 1;
			}
    else if ( inst->internal.fb.DevUnlink_0.status == fiERR_DEVICE_INVALID_HANDLE )
    {
     inst->internal.fb.DevUnlink_0.enable = 0;
     inst->internal.src_handle = 0;
     inst->internal.sc.bNext = 1;
    }
    else if ( inst->internal.fb.DevUnlink_0.status == ERR_FUB_BUSY )
    {

    }
			break;

		case 8:

			brsstrcpy((UDINT)&inst->internal.sc.StepName,(UDINT)&("DevUnlink - destination"));

			inst->internal.fb.DevUnlink_0.enable = 1;
			inst->internal.fb.DevUnlink_0.handle = inst->internal.dest_handle;

			DevUnlink(&inst->internal.fb.DevUnlink_0);

			if (inst->internal.fb.DevUnlink_0.status == ERR_OK)
			{
				inst->internal.fb.DevUnlink_0.enable = 0;
				inst->internal.dest_handle = 0;
    inst->send = 0;
				inst->internal.sc.bLast = 1;
			}
   else if ( inst->internal.fb.DevUnlink_0.status == fiERR_DEVICE_INVALID_HANDLE )
   {
    inst->internal.fb.DevUnlink_0.enable = 0;
    inst->internal.src_handle = 0;
    inst->send = 0;
    inst->internal.sc.bLast = 1;
   }
   else if ( inst->internal.fb.DevUnlink_0.status == ERR_FUB_BUSY )
   {

   }
			break;

		default:

			break;
	}

}
else {

	inst->active = 0;
	inst->internal.sc.step = 0;

	inst->internal.fb.DirRead_0.enable = 0;
	DirRead(&inst->internal.fb.DirRead_0);

	inst->internal.fb.DirInfo_0.enable = 0;
	DirInfo(&inst->internal.fb.DirInfo_0);

	inst->internal.fb.FileDelete_0.enable = 0;
	FileDelete(&inst->internal.fb.FileDelete_0);

	inst->internal.fb.FileCopy_0.enable = 0;
	FileCopy(&inst->internal.fb.FileCopy_0);

	inst->internal.fb.Devlink_0.enable = 0;
	DevLink(&inst->internal.fb.Devlink_0);

}

}
```

#### SKTcpClientSC.c - SKTcpClientSC
```c
/*************************************************************
*
*         projekt: SKTcp - Panasonic
*
*         autor: Ing. Milan Jun
*         company: B+R Automatizace spol. s r.o.
*         date: 21.09.2020
*
*/

#include <bur/plctypes.h>
#ifdef __cplusplus
	extern "C"
	{
#endif
	#include "SKTcp.h"
#ifdef __cplusplus
	};
#endif

/* SKTcpClientSC */
unsigned char SKTcpClientSC(struct SKTcpClientSC_Type* sc)
{

	if ( sc->bNext == 1 ) {

		sc->bNext = 0;
		sc->bRepeat = 0;
		sc->edge = 0;
		sc->step++;

	}

 if ( sc->bLast == 1 ) {

  sc->bLast = 0;
  sc->bRepeat = 0;
  sc->edge = 0;
  sc->step = 0;

 }

 if ( sc->bJump == 1 ) {

  sc->bJump = 0;
  sc->bRepeat = 0;
  sc->edge = 0;

 }

	TON(&sc->idle_time);
	TON(&sc->alarm_time);

	return 0;

}
```

### Library Logical/Libraries/RFID (IEC, version 3.10.0) - A new source library

#### RFID.typ - Exported data types
```iecst
(********************************************************************
 * COPYRIGHT -- Bernecker + Rainer
 ********************************************************************
 * Library: RFID
 * File: RFID.typ
 * Author: houx
 * Created: March 25, 2009
 ********************************************************************
 * Data types of library RFID
 ********************************************************************)

TYPE
	Info : 	STRUCT
		ID : UDINT;
		Type : UDINT;
		StackLevel : UDINT;
	END_STRUCT;
	status : 	STRUCT
		GetUsbList : UINT;
		GetUsbNode : UINT;
		ReleaseBuffer : UINT;
		XOPEN : UINT;
		WRITE : UINT;
		READ : UINT;
		GetBuffer : UINT;
		RoBuffer : UINT;
	END_STRUCT;
	usbDevice : 	STRUCT
		vendorID : UDINT;
		productId : UDINT;
		bcdDevice : UDINT;
	END_STRUCT;
END_TYPE

(**)
```

#### RFID.var - Exported constants
```iecst
(********************************************************************
 * COPYRIGHT -- Bernecker + Rainer
 ********************************************************************
 * Library: RFID
 * File: RFID.var
 * Author: houx
 * Created: March 25, 2009
 ********************************************************************
 * Constants of library RFID
 ********************************************************************)
VAR CONSTANT
	REG1 : USINT := 1;
	REG2 : USINT := 2;
	REG4 : USINT := 4;
	REG5 : USINT := 5;
	REG6 : USINT := 6;
	REG8 : USINT := 8;
	REG9 : USINT := 9;
	REG11 : USINT := 11;
	REG14 : USINT := 14;
	REG13 : USINT := 13;
	REG12 : USINT := 12;
	REG10 : USINT := 10;
	REG7 : USINT := 7;
	REG15 : USINT := 15;
	REG16 : USINT := 16;
	REG19 : USINT := 19;
	REG18 : USINT := 18;
	REG17 : USINT := 17;
	REG20 : USINT := 20;
	REG25 : USINT := 25;
	REG26 : USINT := 26;
	REG28 : USINT := 28;
	READ : USINT := 2;
	WRITE : USINT := 1;
	REG30 : USINT := 30;
	REG33 : USINT := 33;
	CLOSE : USINT := 100;
	REG32 : USINT := 32;
	REG31 : USINT := 31;
	SEARCHTP : USINT := 1;
	SEARCHTPLIST : USINT := 0;
	REG29 : USINT := 29;
	REG27 : USINT := 27;
	STACKWRITE : USINT := 5;
	TRANSPONDER_VENDOR_ID : UINT := 1659;
	TYPEREAD : USINT := 2;
	TRANSPONDER_PRODUCT_ID : UINT := 8963;
	TYPEWRITE : USINT := 1;
	TRANSPONDER_BCD : UINT := 768;
	STACKREAD : USINT := 6;
	REG24 : USINT := 24;
	RW : USINT := 1;
	REG23 : USINT := 23;
	REG22 : USINT := 22;
	REG21 : USINT := 21;
	OPEN : USINT := 0;
	IDWRITE : USINT := 3;
	IDREAD : USINT := 4;
	rfidError_lock_wrongType : UDINT := 41;
	rfidError_password_wrongType : UDINT := 61;
	rfidError_stacklevel_failed : UDINT := 23;
	rfidError_unlock_failed : UDINT := 52;
	rfidError_unlock_wrongType : UDINT := 51;
	rfidError_tag_failed : UDINT := 21;
	rfidError_crc_failed : USINT := 31;
	rfidError_id_failed : UDINT := 22;
	rfidError_write_failed : UDINT := 83;
	rfidError_write_wrongRegNr : UDINT := 82;
	rfidError_write_wrongType : UDINT := 81;
	rfidError_read_wrongRegNr : UDINT := 72;
	rfidError_read_wrongType : UDINT := 71;
	rfidError_rf_failed : UDINT := 11;
	rfidError_read_failed : UDINT := 73;
	rfidError_password_failed : UDINT := 62;
	rfidError_lock_failed : UDINT := 42;
	DATAREAD : USINT := 3;
	REG3 : USINT := 3;
END_VAR
```
